# B&R Automation Studio project 8238 (part 24)

#### vc.ab
```automation-basic
;----------------------------------------------------
;Sequence 1 - SVC1 Vertical conveyor 1 D[900 + mySeq]
;----------------------------------------------------

PROGRAM _INIT
myHttp = 6
END_PROGRAM

PROGRAM _CYCLIC

;Inputs
myVC					    = 1 	;Vertical conveyor number
mySeq					    = 31		;Sequence number
myBag						= 319
myBufferBag					= 360
myIO						= 31
myZone						= 1
myFullLine					= 48
myFullBuffBag				= Line[myFullLine].FirstBag
myFullRelLine				= 0
myFullRelBag				= 0//Line[myFullRelLine].LastBag
myEmptyRelLine				= 0
myEmptyRelBag				= 0
myWeighBag					= 482

//Calculate weight
raw = DINT(AI1223[1])
raw = (raw * 2000)
Bag[myWeighBag].Cat = 1
IF (raw > 0) THEN
	Bag[myWeighBag].Wgt = UINT(raw/32767)
ELSE
	Bag[myWeighBag].Wgt = 0
ENDIF

IF (Bag[myWeighBag].Bid = 0) AND (BidStn > 0) THEN
	Bag[myWeighBag].Bid =  BidStn
	BidStn = 0
ENDIF

RB_PosnName[myVC].Name[1]	= posnNameHighLevelBagOut
RB_PosnName[myVC].Extra[1]	= posnExtraNone
RB_PosnName[myVC].Name[2]	= posnNameHighLevelBagIn
RB_PosnName[myVC].Extra[2]	= posnExtraNone
RB_PosnName[myVC].Name[3]	= posnNameLowLevelBagOut
RB_PosnName[myVC].Extra[3]	= posnExtraNone
RB_PosnName[myVC].Name[4]	= posnNameLowLevelBagIn
RB_PosnName[myVC].Extra[4]	= posnExtraNone

stopZone 		= Std.HaltSysZone[myZone] ;OR ;ZoneControl[myZone].requestAccess
;;ZoneControl[myZone].sequenceRunning[mySeq] = FALSE

I_BagAtOutbuffer			= FALSE
I_OutbufferOpen				= FALSE

;Set rail alignment direction
RailAlignPosn[1] 			= AlignRelease 	;Empty In
RailAlignPosn[2] 			= AlignReceive 	;Full Out
RailAlignPosn[3] 			= AlignRelease 	;Empty Out
RailAlignPosn[4] 			= AlignReceive 	;Full In
RailAlignPosn[5] 			= AlignNone
RailAlignPosn[6] 			= AlignNone

;Sequence Inputs
I_BagOnCarr					= X[myIO].X05
I_BagArriveCarr				= X[myIO].X04
I_PowerSave					= FALSE
I_BagAtFullBuffer			= Line[myFullLine].BufferProximity
I_BagReleased				= X[myIO + 1].X02// Released at high level
;BulkMode = NOT I_AutoMode

O_OpenBuffer					= FALSE
O_OpenCarrStop					= FALSE
O_Lamp                      	= FALSE
O_OpenFullBagBuffer				= FALSE

Request.VC[myVC]				= FALSE
Request.VC_HighLevel[myVC]  	= FALSE
Request.VC_LowLevel[myVC]	    = FALSE
RequestRel.VC_HighLevel[myVC]	= FALSE
RequestRel.VC_LowLevel[myVC]	= FALSE

EnableRel.PN[31]				= FALSE

;Lifting
strcpy(ADR(LiftIn.sDevice),ADR("SS1.IF1"))
strcpy(ADR(LiftIn.sParTblName),ADR("Param_1_5k"))
LiftIn.Node					= (10 + myVC)

LiftIn.DisableDrive			= FALSE
LiftIn.DoRef 				= FALSE
LiftIn.JogForwards 			= FALSE
LiftIn.JogReverse 			= FALSE
LiftIn.EStop				= Std.HaltSysZone[myZone]
LiftIn.PosnReq				= 0
LiftIn.MaxSpeed				= RB_Posn[myVC].Lift.MaxSpeed
LiftIn.PowerSave 			= FALSE
LiftIn.I_ForwardLimitOk		= X[myIO + 1].X01 	;Top limit   	- Do NOT Change to N.O.
LiftIn.I_ReverseLimitOk		= X[myIO + 1].X03	;Bottom limit	- Do NOT Change to N.O.
LiftIn.I_RefPosn			= X[myIO + 1].X04
LiftIn.I_RailOkRelease		= X[myIO].X07
LiftIn.I_RailOkReceive		= X[myIO].X06

LiftOut						= RB[myVC].Lift.SeqOut ;Copy drive outputs to local

;Shared Lift & Rotate
DisableDrive				= FALSE
RunMotor 					= FALSE
RunPosition					= 0

;Clear Interlock Signals
LOOP Posn = 1 TO 5 DO
	VCiLock[myVC].Posn[Posn].EnabSend 	= FALSE
ENDLOOP

Alarm[mySeq].Name 			= 0
Alarm[mySeq].Bag			= myBag
Alarm[mySeq].Beacon			= TRUE
Alarm[mySeq].Extra			= 0
Alarm[mySeq].Time			= 6000

;Setup Sequence
STEP = D[900 + mySeq]
;Setup Pulse contact
PLS = (STEP <> LASTSTEP)
LASTSTEP = STEP

;Sequence
IF (STEP = 0) THEN
	;Disabled
	DisableDrive 	= TRUE
ENDIF

;Combine Lift and Rotate into a single variable
DrivesReady		= LiftOut.RefComplete
DriveDisabled 	= (NOT PLS AND LiftOut.DriveDisabled) OR DebugMode
PosnOk	 		= (NOT PLS AND LiftOut.PosnOk)
RailOkReceive	= LiftIn.I_RailOkReceive
RailOkRelease	= LiftIn.I_RailOkRelease

;Power Save mode
IF I_PowerSave THEN
	LiftIn.PowerSave 	= TRUE
	LiftIn.MaxSpeed		= 300
ENDIF

;Carriage Empty Decide what to do next.
IF (STEP = 1) THEN
	;Cycle Count
    ;ZoneControl[myZone].sequenceRunning[mySeq] = TRUE
	IF PLS THEN
		CycleCount 						= CycleCount + 1
		RB_Perm[myVC].Lift.CycleCount 	= RB_Perm[myVC].Lift.CycleCount + 1
	ENDIF
	IF NOT Std.HaltSysZone[myZone]  THEN
		IF (CycleCount >= 500) THEN
			;If Referencing required then set 'Do Reference'
			;Put the sequence to a position step to enable the carriage
			;to retuen to the correct place after referencing
			LiftIn.DoRef 	= TRUE
			CycleCount 		= 0
		ELSE
			INC Count[mySeq]
			D[900 + mySeq] = 2
		ENDIF
	ENDIF
ENDIF

;Step 2. Move to empty bag in high level.....
IF (STEP = 2) THEN
	RunPosition	= POS_EMPTY_BAG_IN
	;ZoneControl[myZone].sequenceRunning[mySeq] = TRUE
	RunMotor	= (NOT Std.HaltSysZone[myZone] AND DrivesReady)
	IF PosnOk THEN
		D[900 + mySeq] = 3
	ENDIF
	IF (NOT Std.HaltSysZone[myZone] AND DrivesReady) THEN
		Alarm[mySeq].Name = almCarriageMoveFault
	ENDIF
ENDIF

GetFullBag	 = (Bag[myFullBuffBag].Cat > 0)
GetEmpty	 = RequestRel.PN[31] //And check lower loop space.

;Decide what to do
TON_10ms((NOT I_BagArriveCarr AND NOT I_BagOnCarr),300,CarriageClear,CarriageClearET)
IF (STEP = 3) THEN
	DisableDrive = TRUE
	IF CarriageClear AND (Bag[myBag].Cat = 0) AND NOT stopZone  THEN
	 	Request.VC[myVC] = TRUE // Tell CP31 that vc is in position..
		IF GetEmpty THEN
			D[900 + mySeq] = 4
		ELSE IF GetFullBag THEN
			D[900 + mySeq] = 9
		ENDIF
	ENDIF
  IF NOT CarriageClear THEN
		Alarm[mySeq].Name = almSwitchFault
	ELSE IF (Bag[myBag].Cat > 0) THEN
		Alarm[mySeq].Name = almBagDataError
	ENDIF
ENDIF

;Enable CP31 to release a bag
IF (STEP = 4) THEN
	DisableDrive = TRUE
    ;ZoneControl[myZone].sequenceRunning[mySeq] = TRUE
	EnableRel.PN[31] = (Bag[myBag].Cat = 0)
	IF (I_BagOnCarr OR I_BagArriveCarr) THEN
		D[900 + mySeq] = 5
	ENDIF
	IF NOT RailOkReceive THEN
		Alarm[mySeq].Name = almRailNotAligned
		Alarm[mySeq].Time = 100
	ENDIF
ENDIF

;Bag settles on carriage
TON_10ms(I_BagOnCarr,300,SettledCarriage,SettledCarriageET)
IF (STEP = 5) THEN
	DisableDrive = TRUE
	IF SettledCarriage AND (Bag[myBag].Cat > 0) AND NOT stopZone AND NOT EnableRel.VC_LowLevel[myVC] THEN
		D[900 + mySeq] = 6
	ELSE IF NOT SettledCarriage	THEN
		Alarm[mySeq].Name = almBagNotSettled
		Alarm[mySeq].Time = 9000
	ELSE IF (Bag[myBag].Cat = 0) THEN
		Alarm[mySeq].Name = ALM_BAG_DATA_ERROR
		Alarm[mySeq].Time = 0
	ENDIF
ENDIF

;Move carriage to empty bag out.
IF (STEP = 6) THEN
	RunPosition	= POS_EMPTY_BAG_OUT
    ;ZoneControl[myZone].sequenceRunning[mySeq] = TRUE
	RunMotor	= (NOT Std.HaltSysZone[myZone] AND DrivesReady)
	IF PosnOk THEN
		D[900 + mySeq] = 7
	ENDIF
	IF (NOT Std.HaltSysZone[myZone] AND DrivesReady) THEN
		Alarm[mySeq].Name = almCarriageMoveFault
	ENDIF
ENDIF

;Request Release
releaseValid = (Bag[myBag].Cat > 0)AND RailOkRelease
IF (STEP = 7) THEN
	DisableDrive = TRUE
	RequestRel.VC_LowLevel[myVC] = releaseValid
	IF EnableRel.VC_LowLevel[myVC] AND releaseValid THEN
		D[900 + mySeq] = 8
	ELSE IF NOT RailOkRelease THEN
		Alarm[mySeq].Name = almRailNotAligned
		Alarm[mySeq].Time = 100
	ELSE IF (Bag[myBag].Cat = 0) THEN
		Alarm[mySeq].Name = ALM_BAG_DATA_ERROR
		Alarm[mySeq].Time = 0
	ENDIF
ENDIF

;STEP 8 release empty bag
IF (STEP = 8) THEN
	DisableDrive = TRUE
	O_OpenCarrStop = releaseValid
	IF (Bag[myBag].Cat = 0) AND NOT EnableRel.VC_LowLevel[myVC] THEN
		IF GetFullBag OR (D[901] > 6) THEN//CHeck if there is a full bag, or the loading unit is releasing before moving back to the top,,
			D[900 + mySeq] = 9
		ELSE
			D[900 + mySeq] = 1
		ENDIF
	ELSE IF releaseValid THEN
		Alarm[mySeq].Name = ALM_BAG_NOT_RELEASED
	ELSE IF NOT RailOkRelease THEN
		Alarm[mySeq].Name = almRailNotAligned
		Alarm[mySeq].Time = 100
	ELSE IF (Bag[myBag].Cat = 0) THEN
		Alarm[mySeq].Name = ALM_BAG_DATA_ERROR
		Alarm[mySeq].Time = 0
	ENDIF
ENDIF

;Step 9. Move to full bag in.....
IF (STEP = 9) THEN
	RunPosition	= POS_FULL_BAG_IN
    ;ZoneControl[myZone].sequenceRunning[mySeq] = TRUE
	RunMotor	= (NOT Std.HaltSysZone[myZone] AND DrivesReady)
	IF PosnOk THEN
		D[900 + mySeq] = 10
	ENDIF
	IF (NOT Std.HaltSysZone[myZone] AND DrivesReady) THEN
		Alarm[mySeq].Name = almCarriageMoveFault
	ENDIF
ENDIF

//Wait for bag at full buffer
TON_10ms(I_BagAtFullBuffer,300,SettledFullBuffer,SettledFullBufferET)
IF (STEP = 10) THEN
	IF SettledFullBuffer AND (Bag[myBag].Cat = 0) AND (Bag[myFullBuffBag].Cat > 0) AND RailOkReceive THEN
		D[900 + mySeq] = 11
	ELSE IF NOT RailOkReceive THEN
		Alarm[mySeq].Name = ALM_RAIL_NOT_ALIGNED
		Alarm[mySeq].Time = 0
	ELSE IF (Bag[myBag].Cat > 0) THEN
		Alarm[mySeq].Name = ALM_BAG_DATA_ERROR
		Alarm[mySeq].Time = 0
	ELSE IF SettledFullBuffer AND (Bag[myFullBuffBag].Cat = 0) THEN
		Alarm[mySeq].Name = ALM_BAG_DATA_ERROR
		Alarm[mySeq].Bag = myFullBuffBag
	ELSE IF NOT SettledFullBuffer AND (Bag[myFullBuffBag].Cat > 0)THEN
		Alarm[mySeq].Name = ALM_BAG_NOT_SETTLED
		Alarm[mySeq].Time = 500
	ENDIF
ENDIF

;Open Full buffer stop
IF (STEP = 11) THEN
	DisableDrive = TRUE
    O_OpenFullBagBuffer = (Bag[myBag].Cat = 0) AND (Bag[myFullBuffBag].Cat > 0);
	IF I_BagOnCarr OR I_BagArriveCarr THEN
		Bag[myBag] = Bag[myFullBuffBag]
		Bag[myFullBuffBag] = Bag[0]
		D[900 + mySeq] = 12
	ENDIF
	IF (Bag[myBag].Cat > 0) THEN
		Alarm[mySeq].Name = ALM_BAG_DATA_ERROR
		Alarm[mySeq].Time = 0
	ELSE IF NOT RailOkReceive THEN
		Alarm[mySeq].Name = almRailNotAligned
		Alarm[mySeq].Time = 100
	ENDIF
ENDIF

;Bag settles on carriage
TON_10ms((STEP = 12) AND I_BagOnCarr AND NOT I_BagArriveCarr,300,SettledCarriage12,SettledCarriage12ET)
TON_10ms(((STEP = 12) AND (Bag[myWeighBag].Wgt < 1250)),600,weightOk,weightOkET)
IF (STEP = 12) THEN
	DisableDrive = TRUE
	IF SettledCarriage12 AND weightOk AND (Bag[myBag].Cat > 0) AND NOT stopZone  THEN
		Bag[myBag].Wgt := Bag[myWeighBag].Wgt;
		D[900 + mySeq] = 13
	ELSE IF NOT weightOk THEN
		Alarm[mySeq].Name = almBagOverWeight
	ELSE IF (Bag[myBag].Cat = 0) THEN
	//	Alarm[mySeq].Name = almBagDataError
	ELSE IF NOT stopZone THEN
		Alarm[mySeq].Name = almBagNotSettled
		Alarm[mySeq].Time = 9000
	ENDIF
ENDIF

;Move carriage to full bag out.
IF (STEP = 13) THEN
	RunPosition	= POS_FULL_BAG_OUT
    ;ZoneControl[myZone].sequenceRunning[mySeq] = TRUE
	RunMotor	= (NOT Std.HaltSysZone[myZone] AND DrivesReady)
	IF PosnOk THEN
		D[900 + mySeq] = 14
	ENDIF
	IF (NOT Std.HaltSysZone[myZone] AND DrivesReady) THEN
		Alarm[mySeq].Name = almCarriageMoveFault
	ENDIF
ENDIF

//Weighing step  Send to Data base. Add to batch...
IF (STEP = 14) THEN
	IF (Bag[myBag].Mis > 0) THEN
		_httpRequest
		IF httpComplete AND NOT EnableRel.VC_HighLevel[myVC] THEN
			myReportStn = 1
			IF (ReportLoading[myReportStn].Cat = 0) THEN
				ReportLoading[myReportStn].Prg := Bag[myBag].Prg;
				ReportLoading[myReportStn].Cat := Bag[myBag].Cat;
				ReportLoading[myReportStn].Cus := Bag[myBag].Cus;
				ReportLoading[myReportStn].Wgt := Bag[myBag].Wgt;
				ReportLoading[myReportStn].Cnt := 0;
				ReportLoading[myReportStn].Stn := myReportStn;
				ReportLoading[myReportStn].Mcn := 0;
				ReportLoading[myReportStn].Bid := Bag[myBag].Bid;
				ReportLoading[myReportStn].Mis := Bag[myBag].Mis;
				ReportLoading[myReportStn].TimeStamp := Bag[myBag].Timestamp;
				D[900 + mySeq] = 15
			ENDIF;
		ELSE
			Alarm[mySeq].Name = ALM_GENERAL_SEQUENCE
		ENDIF
	ELSE
		Alarm[mySeq].Name = ALM_BAG_DATA_ERROR
	ENDIF
ELSE
	httpComplete = 0
	HTTP_Comm[myHttp].Status = HTTP_COMM_STATUS_DISABLED
ENDIF;

DataValid = (Bag[myBag].Cat > 0)// AND (Bag[myFullRelBag].Cat = 0))
;check data valid
IF (STEP = 15) THEN
	DisableDrive = TRUE
	RequestRel.VC_HighLevel[myVC] = DataValid AND RailOkRelease AND NOT stopZone
	IF  EnableRel.VC_HighLevel[myVC] THEN
		D[900 + mySeq] = 16
	ELSE IF (Bag[myBag].Cat = 0) THEN
	//	Alarm[mySeq].Name = almBagDataError
	ELSE IF NOT RailOkRelease THEN
		Alarm[mySeq].Name = almRailNotAligned
		Alarm[mySeq].Time = 100
	ENDIF
ENDIF

;STEP 15 Open Stops release full bag
IF (STEP = 16) THEN
	DisableDrive = TRUE
    ;ZoneControl[myZone].sequenceRunning[mySeq] = TRUE
	O_OpenCarrStop = EnableRel.VC_HighLevel[myVC] AND RailOkRelease
	IF (NOT EnableRel.VC_HighLevel[myVC] OR I_BagReleased) AND (Bag[myBag].Cat = 0) THEN
		D[900 + mySeq] = 1
	ENDIF
	IF NOT stopZone THEN
		IF NOT EnableRel.VC_HighLevel[myVC]  AND (Bag[myBag].Cat > 0) THEN
			Alarm[mySeq].Name = ALM_BAG_DATA_ERROR
		ELSE IF NOT RailOkRelease THEN
			Alarm[mySeq].Name = almRailNotAligned
			Alarm[mySeq].Time = 100
		ENDIF
	ENDIF
ENDIF

;-----------------------------------------------------------
;No Changes required below here except PLC outputs at bottom
;-----------------------------------------------------------

;Positions Required
IF (RunPosition > 0) THEN
	LiftIn.PosnReq		= RB_Posn[myVC].Lift.Posn[RunPosition]
	LiftIn.RailAlign 	= RailAlignPosn[RunPosition]

	RotateIn.PosnReq	= RB_Posn[myVC].Rotate.Posn[RunPosition]
	RotateIn.RailAlign 	= RailAlignPosn[RunPosition]
ELSE
	LiftIn.PosnReq		= 0
	LiftIn.RailAlign	= 0

	RotateIn.PosnReq	= 0
	RotateIn.RailAlign 	= 0
ENDIF

;Bag detected on carriage at wrong time during operation
IF ((RunPosition > 0) AND RunMotor) THEN
	IF I_BagArriveCarr THEN
		LiftIn.EStop	= TRUE ;Force Quickstop
		RunPosition		= 0
		RunMotor		= FALSE
		D[900 + mySeq] 	= 97
	ELSE IF (I_BagOnCarr AND (RailAlignPosn[RunPosition] = AlignReceive)) THEN
		LiftIn.EStop	= TRUE ;Force Quickstop
		RunPosition		= 0
		RunMotor		= FALSE
		D[900 + mySeq] 	= 98
	ENDIF
ENDIF
IF (STEP = 97) THEN
	DisableDrive = TRUE
	Alarm[mySeq].Name 	= almDisableSequence
	Alarm[mySeq].Time			= 100
ENDIF
IF (STEP = 98) THEN
	DisableDrive = TRUE
	Alarm[mySeq].Name 	= almDisableSequence
	Alarm[mySeq].Time			= 100
ENDIF

;Position Setup
TON_10ms(VCHeartBeat = D[84],100,VCActionDisabled,VCActionDisabledET)
IF (STEP = 99) THEN

	RB_Posn[myVC].Lift.OperationMode 	= 1 ;Manual Position Setup
	RB_Posn[myVC].Rotate.OperationMode 	= 1 ;Manual Position Setup

	;Read values sent from TrackView
	VCIndex 	= D[81]
	VCMode 		= D[82]
	VCAction 	= D[83]
	VCHeartBeat = D[84]

	IF ((VCIndex = myVC) AND NOT VCActionDisabled) THEN

		IF (VCMode = ModeReference) THEN
			LiftIn.DoRef 			= TRUE
			RotateIn.DoRef 			= TRUE
		ELSE IF (VCMode = ModeManualMove) THEN
			LiftIn.JogForwards 		= (VCAction = ActionMoveUp)
			LiftIn.JogReverse 		= (VCAction = ActionMoveDown)
			RotateIn.JogReverse		= (VCAction = ActionMoveLeft)
			RotateIn.JogForwards	= (VCAction = ActionMoveRight)
		ELSE IF (VCMode = ModePosnTune) THEN
			AutoTuneSequence		= 1
			AutoTunePosition		= VCAction
		ELSE IF (VCMode = ModeMovePosn) THEN
			RunMotor				= (NOT Std.HaltSysZone[myZone] AND DrivesReady); AND ;PositionSetup)
			LiftIn.MaxSpeed 		= 200
			RotateIn.MaxSpeed 		= 200
			IF (VCAction = 100) THEN
				LiftIn.PosnReq 		= RB_Posn[myVC].Lift.RefOffset
				RotateIn.PosnReq 	= RB_Posn[myVC].Rotate.RefOffset
			ELSE
				LiftIn.PosnReq		= RB_Posn[myVC].Lift.Posn[VCAction]
				RotateIn.PosnReq	= RB_Posn[myVC].Rotate.Posn[VCAction]
			ENDIF
		ENDIF

	ENDIF

	;Auto Position Tune Sequnece
	;---------------------------
	IF (AutoTuneSequence = 1) THEN
		;Wait for release of Autotune Button / Command
		IF (VCMode <> ModePosnTune) THEN
			AutoTuneSequence = 2
		ENDIF
	ELSE IF (AutoTuneSequence = 2) THEN
		;Check if rail Aligned
		Aligned = (((RailAlignPosn[AutoTunePosition] = AlignReceive) AND LiftIn.I_RailOkReceive) OR ((RailAlignPosn[AutoTunePosition] = AlignRelease) AND LiftIn.I_RailOkRelease))
		;Begin Lift Tune
		IF Aligned THEN
			LiftIn.AutoTunePosn		= AutoTunePosition
			LiftIn.AutoTuneReceive 	= (RailAlignPosn[AutoTunePosition] = AlignReceive)
			IF (LiftOut.AutoTunePosn = AutoTunePosition) THEN
				AutoTuneSequence = 3
			ENDIF
		ELSE
			AutoTuneSequence = 0 ;Cancel Auto Tune
		ENDIF
	ELSE IF (AutoTuneSequence = 3) THEN
		;Wait for Lift to complete Tune
		IF (LiftOut.AutoTunePosn = 0) THEN
			AutoTuneSequence = 4
		ENDIF
	ELSE IF (AutoTuneSequence = 4) THEN
		;Move to new position
		LiftIn.AutoTunePosn		= 0 ;Cancel Tune
		RunMotor				= (NOT Std.HaltSysZone[myZone] AND DrivesReady); AND ;PositionSetup)
		LiftIn.MaxSpeed 		= 200
		RotateIn.MaxSpeed		= 0  ;Don't allow rotate to move
		LiftIn.PosnReq			= RB_Posn[myVC].Lift.Posn[AutoTunePosition]
		RotateIn.PosnReq		= 0
		IF LiftOut.PosnOk THEN
			AutoTuneSequence = 5
		ENDIF
	ELSE IF (AutoTuneSequence = 5) THEN
		;Begin Rotate Tune
		RotateIn.AutoTunePosn 		= AutoTunePosition
		RotateIn.AutoTuneReceive 	= (RailAlignPosn[AutoTunePosition] = AlignReceive)
		IF (RotateOut.AutoTunePosn = AutoTunePosition) THEN
			AutoTuneSequence = 6
		ENDIF
	ELSE IF (AutoTuneSequence = 6) THEN
		;Wait for Rotate to complete Tune
		IF (RotateOut.AutoTunePosn = 0) THEN
			AutoTuneSequence = 7
		ENDIF
	ELSE IF (AutoTuneSequence = 7) THEN
		;Move to new position
		RotateIn.AutoTunePosn	= 0 ;Cancel Tune
		RunMotor				= (NOT Std.HaltSysZone[myZone] AND DrivesReady); AND ;PositionSetup)
		LiftIn.MaxSpeed 		= 0
		RotateIn.MaxSpeed		= 200
		LiftIn.PosnReq			= 0
		RotateIn.PosnReq		= RB_Posn[myVC].Rotate.Posn[AutoTunePosition]
		IF RotateOut.PosnOk THEN
			AutoTuneSequence = 0
		ENDIF
	ENDIF

ELSE
	;Set Operation mode to Normal
	RB_Posn[myVC].Lift.OperationMode 	= 0
	RB_Posn[myVC].Rotate.OperationMode 	= 0
	;Cancel Auto Tune
	AutoTuneSequence 					= 0
	LiftIn.AutoTunePosn 				= 0
	RotateIn.AutoTunePosn 				= 0
ENDIF

;Lift Drive Alarms
IF (LiftOut.Status = FC302_SEQ_RefNotFound) THEN
	Alarm[mySeq].Name = almLiftRefNotFound
	Alarm[mySeq].Time = 10
ELSE IF (LiftOut.Status = FC302_SEQ_ParameterError) THEN
	Alarm[mySeq].Name = almLiftParameterError
	Alarm[mySeq].Time = 10
ELSE IF (LiftOut.Status = FC302_SEQ_RefSwitchFault) THEN
	Alarm[mySeq].Name = almLiftRefSwitchFault
	Alarm[mySeq].Time = 10
ELSE IF (LiftOut.Status = FC302_SEQ_ReleaseSwitchFault) THEN
	Alarm[mySeq].Name = almReleaseSwitchFault
	Alarm[mySeq].Time = 10
ELSE IF (LiftOut.Status = FC302_SEQ_ReceiveSwitchFault) THEN
	Alarm[mySeq].Name = almReceiveSwitchFault
	Alarm[mySeq].Time = 10
ELSE IF (LiftOut.Status = FC302_SEQ_RailNotAligned) THEN
	Alarm[mySeq].Name = almReleaseSwitchFault
	Alarm[mySeq].Time = 10
ENDIF

;Inputs to drive control sequence
LiftIn.Run			     	= RunMotor
LiftIn.DisableDrive 	= DisableDrive
RB[myVC].Lift.SeqIn 	= LiftIn 	;Copy local to drive inputs

TON_10ms(NOT Std.HaltSysZone[myZone],100,HaltSysZoneClear,HaltSysZoneClearET)	; Safe zone
OpenStopEnabled = (HaltSysZoneClear AND LiftOut.DriveDisabled)

;-----------------------------------
;PLC Outputs - adjust to suit system
;-----------------------------------
Y[22].Y05 = (RailOkReceive AND ((STEP = 11) OR (STEP = 12)) AND DriveDisabled)  ; Safety Stop Low level
Y[myIO + 1].Y05 = (RailOkReceive AND ((STEP = 3) OR (STEP = 4) OR (STEP = 5)) AND DriveDisabled) ; Safety Stop High level
Y[4].Y06 		= (O_OpenCarrStop AND RailOkRelease AND OpenStopEnabled AND DriveDisabled)

Line[myFullLine].BufferStop := O_OpenFullBagBuffer

;Don't allow forcing of carriage movement and carriage stop
YForceDisable[myIO].Y07 	= TRUE
YForceDisable[myIO].Y08 	= TRUE
;YForceDisable[6].Y04 	= TRUE

;Alarms
TimerAlarm.IN 		= NOT PLS AND (Alarm[mySeq].Name > 0)
TimerAlarm.PT 		= Alarm[mySeq].Time
TimerAlarm FUB TON_10ms()
Alarm[mySeq].On 	= TimerAlarm.Q
Alarm[mySeq].ET 	= TimerAlarm.ET

END_PROGRAM
```

#### _httpRequest.st
```iecst
ACTION _httpRequest:

	CASE HTTP_Comm[myHttp].Status OF

		HTTP_COMM_STATUS_DISABLED:

			//Build Request String..
			requestURL := HTTP_IF_CALL_USP_NOREPLY_URL;
			itoa(Bag[myBag].Mis,ADR(batchString));
			itoa(Bag[myWeighBag].Wgt,ADR(weightString));
			//Bag[myBag].Wgt := Bag[myWeighBag].Wgt;

			requestData := CONCAT(HTTP_POST_BATCH_UPDATE_DRY_WGT,'@BatchID_Int=');
			requestData := CONCAT(requestData,batchString);
			requestData := CONCAT(requestData,',@DryWeight=');
			requestData := CONCAT(requestData,weightString);

			HTTP_Comm[myHttp].Command.Method := httpMETHOD_POST;
			HTTP_Comm[myHttp].Command.Cmd_URL.Adr := ADR(requestURL);
			HTTP_Comm[myHttp].Command.Cmd_URL.Size := LEN(requestURL);
			HTTP_Comm[myHttp].Command.Body_Data.Adr := ADR(requestData);
			HTTP_Comm[myHttp].Command.Body_Data.Size := strlen(ADR(requestData));
			HTTP_Comm[myHttp].Command.ResponseData.Adr := 0;
			HTTP_Comm[myHttp].Command.ResponseData.Size := 0;
			HTTP_Comm[myHttp].Status := HTTP_COMM_STATUS_ACTIVE_WAIT_BUF;

		HTTP_COMM_STATUS_ACTIVE_WAIT_BUF:
		//Command is sent to ring buffer.
		HTTP_COMM_STATUS_IN_BUFFER:
		//Command recieved and in ring buffer
		HTTP_COMM_STATUS_IN_PROCESS:
		//Command being processed by httpClient.
		HTTP_COMM_STATUS_COMPLETE:
			httpComplete := 1;
			//HTTP_Comm[myHttp].Status := HTTP_COMM_STATUS_DISABLED;
		HTTP_COMM_STATUS_ERROR: // Go to next index
			HTTP_Comm[myHttp].Status := HTTP_COMM_STATUS_DISABLED;

	END_CASE;

END_ACTION
```

### Program Logical/Robo_Drive_Control/Lift_v8_1 (IEC, version 8.00.2)

#### Lift.var - Local variables
```iecst
(********************************************************************
 * COPYRIGHT --
 ********************************************************************
 * Program: PosnVC
 * File: PosnVC.var
 * Author: D.Jefferys
 * Created: February 12, 2009
 ********************************************************************
 * Local variables of program PosnVC
 ********************************************************************)
VAR
	AutoNewPosn : DINT;
	AutoPosnDiff : DINT;
	AutoSavedBottom : DINT;
	AutoSavedTop : DINT;
	CANopenNMT_0 : CANopenNMT;
	DisableDrive : BOOL;
	DistRemain : DINT;
	EnableDrive : BOOL;
	EnableForwards : BOOL;
	EnableReference : BOOL;
	EnableReverse : BOOL;
	EnableTune : BOOL;
	FC302_ReadParam_0 : FC302_ReadParam;
	FC302_ReadParamTbl_0 : FC302_ReadParamTbl;
	FC302_ReadSTW_0 : FC302_ReadSTW;
	FC302_WriteCTW_0 : FC302_WriteCTW;
	FC302_WriteParam_0 : FC302_WriteParam;
	I_InPosition : BOOL;
END_VAR
VAR RETAIN
	idx : UINT;
END_VAR
VAR
	LimitsOk : BOOL;
	ManualControl : BOOL;
	MaxHz : UINT;
	MonitorIndex : UINT := 0;
	MonitorSubIndex : USINT;
	MotorNomHz : UINT;
	myRead : UDINT;
	myStatus : UINT;
	node : USINT;
	ParameterEnable : BOOL;
	PosnDiff : DINT;
	PosnValid : BOOL;
	PowerSave : BOOL;
	QuickStop : BOOL;
	RailAligned : BOOL;
	RampDist : REAL;
	RampFactor : REAL;
	RampTime : UINT;
	Referencing : BOOL;
	ReleaseSwitchOk : BOOL := FALSE;
	ReceiveSwitchOk : BOOL := FALSE;
	RequiredHz : UINT;
	ResetTrip : BOOL;
	RunSpeed : REAL;
	RunTask : BOOL;
	SavedBottom : DINT;
	SavedPosition : DINT;
	SavedTop : DINT;
	ScanClock : TIME;
	ScanCount : UINT;
	ScanLastClock : TIME;
	ScanNow : TIME := T#0ms;
	sDevice : STRING[12];
	SlowWindow : DINT;
	sTableName : STRING[10];
	STEP : UINT;
	StopDist : DINT;
	StopFactor : REAL;
	TableTooLarge : BOOL;
	TaskName : STRING[11];
	TaskNameID : UINT;
	TaskNameLen : UINT;
	TON_10ms_PastRef : TON_10ms;
	TON_10ms_Restart : TON_10ms;
	TON_10ms_Retry : TON_10ms;
	WriteIndex : UINT;
	WriteListLength : UINT;
	JogHz : UINT;
	TmrJog : TON_10ms;
	AlignSwitchCheck : BOOL;
	AlignSwitchesOk : BOOL;
	mySlowWindow : DINT;
	myDist : DINT;
	RefSpeed : UINT;
	CountCardFailedPLS : BOOL;
	RetryCount : UINT;
	I_RefPosnPLS : BOOL;
	AutoRefTolerance : DINT;
	Debug_PositionErrorCount : UDINT;
	PositionErrorLastValue : ARRAY[0..100] OF DINT;
	IndexPostion : UINT;
	Debug_CycleCount : UDINT;
	DebugLastActual : DINT;
	DebugRef : DINT;
	PositionError : DINT;
	TestValue : DINT;
	TestResult : DINT;
END_VAR
```

#### Lift.ab - Cyclic code
```automation-basic
;--------------------------------------
;Lift Drive Control - Original 2 Column
;--------------------------------------

;Version 1.00 23/02/2009 D.J. First Issue
;Version 2.00 03/11/2010 D.J. Changed RB to RB (Robo)
;Version 3.00 04/12/2010 D.J. New distance calculation by using encoder pulses for 1 meter
;Version 4.00 04/03/2011 D.J. Set RunHz to 0 when not on step 30
;Version 5.00 08/01/2013 T.R Add module OK to monitor Counter Card and force step 0 after error/powerup..Increased Param Count for Brake contact monitoring. Force init values when 0.
;Version 5.01 12/03/2013 T.R Change function of module OK monitoring to always restart seq after fail due to power cycles on remote panels.
;Version 6.01 			T.R Add Auto Reference function
;Version 6.02 27/11/2015 TR. Add Correct comments,
;Version V8 -- TR Send QS command when enable is off due to DANFOSS issues.

PROGRAM _INIT

 	;Set array index with each init call
	idx  = 0

	TaskNameID = ST_name(0,ADR(TaskName),0)

	IF (TaskNameID = 0) THEN
		TaskNameLen = strlen(ADR(TaskName))
		idx 		= UINT(atoi(ADR(TaskName) + (TaskNameLen - 1)))
	ENDIF

	RunTask = (idx > 0) and (idx <= (SIZEOF(RB)/SIZEOF(RB[0])))

	IF RunTask THEN

		;Calculate in future for different arrangements
		;----------------------------------------------

		;New calculation based on measuring the pulsed for 1000 mm of Travel
		;-------------------------------------------------------------------

		;Pulses per meter = 122864.6
		;My Ratio (Gearbox and Cog combined) = 4096 / 122.8646 = 33.3375
		;mm/minute 				= Motor Nominal Speed 1500 * My Ratio = 50006.25
		;mm/sec @ 50 Hz 		= 833.4375
		;mm/Hz 	833.4375 / 50 	= 16.6687

		RB[idx].Lift.PulsePer10th_mm = REAL(12.2865)
		RB[idx].Lift.mmPerHz = 16.6687
		;Force Init value if 0
		IF RB_Posn[idx].Lift.RefOffset = 0 THEN
			RB_Posn[idx].Lift.RefOffset = 20000 ; 2metres
		ENDIF
		IF RB_Posn[idx].Lift.MaxSpeed = 0 THEN
			RB_Posn[idx].Lift.MaxSpeed = 200
		ENDIF

		// Temp to force input parameters.

		strcpy(ADR(RB[idx].Lift.SeqIn.sDevice),ADR("SL1.IF3"))
		strcpy(ADR(RB[idx].Lift.SeqIn.sParTblName),ADR("Param_1_5k"))
		RB[idx].Lift.SeqIn.Node := 10 + USINT(idx);
		RB[idx].Lift.ModuleOK := TRUE
		// END

	ENDIF

	STEP 					= 0
	RB[idx].Lift.SeqStep	= 0
	RetryCount				= 0

END_PROGRAM
PROGRAM _CYCLIC

	;----
	;Lift
	;----

	myStatus = FC302_SEQ_OK

	;CAN node, Parameter Table Name and IF address
	node 	= RB[idx].Lift.SeqIn.Node
	strcpy(ADR(sTableName),ADR(RB[idx].Lift.SeqIn.sParTblName))
	strcpy(ADR(sDevice),ADR(RB[idx].Lift.SeqIn.sDevice))

	RB[idx].Lift.SeqIn.I_RefPosn  = X[30 + (idx * 2)].X04

	;Read drive status
	FC302_ReadSTW_0.StatusWord = RB[idx].Lift.CAN.StatusWord
	FC302_ReadSTW_0 FUB FC302_ReadSTW()
	RB[idx].Lift.STW = FC302_ReadSTW_0.STW

	;Clear control word - drive stopped
	RB[idx].Lift.CTW.ExtRefSelectionLSB 	= FALSE
	RB[idx].Lift.CTW.ExtRefSelectionMSB 	= FALSE
	RB[idx].Lift.CTW.DC_Brake				= FALSE
	RB[idx].Lift.CTW.Coasting				= FALSE
	RB[idx].Lift.CTW.QuickStop				= FALSE
	RB[idx].Lift.CTW.HoldOutputFreq			= FALSE
	RB[idx].Lift.CTW.RampStopStart			= FALSE
	RB[idx].Lift.CTW.ResetTrip				= ResetTrip
	RB[idx].Lift.CTW.Jog					= FALSE
	RB[idx].Lift.CTW.RampSelection			= FALSE
	RB[idx].Lift.CTW.DataValid				= TRUE
	RB[idx].Lift.CTW.Relay01Active			= FALSE
	RB[idx].Lift.CTW.Relay02Active			= FALSE
	RB[idx].Lift.CTW.ParaSetUpLSB			= FALSE
	RB[idx].Lift.CTW.ParaSetUpMSB			= FALSE
	RB[idx].Lift.CTW.Reverse				= FALSE

	RB[idx].Lift.RunForwards				= FALSE
	RB[idx].Lift.RunReverse					= FALSE
	RB[idx].Lift.CAN.TargetVelocity			= 0
	RB[idx].Lift.RunFreq 					= 0
	RB[idx].Lift.SeqOut.RefComplete 		= FALSE
	RB[idx].Lift.SeqOut.PosnOk				= FALSE
	RB[idx].Lift.SeqOut.DriveDisabled		= FALSE
	Referencing								= FALSE
	DisableDrive 							= (RB[idx].Lift.SeqIn.DisableDrive OR RB[idx].Lift.SeqIn.EStop OR NOT RB[idx].Lift.STW.DriveReady OR NOT RB[idx].Lift.ModuleOK)
	LimitsOk								= (RB[idx].Lift.SeqIn.I_ForwardLimitOk AND RB[idx].Lift.SeqIn.I_ReverseLimitOk)
	ManualControl							= (RB_Posn[idx].Lift.OperationMode = 1)

	;Init var ensure not lost if no Init
	RB[idx].Lift.PulsePer10th_mm 			= REAL(12.2865)
	RB[idx].Lift.mmPerHz 					= 16.6687

	;Current Position
	RB[idx].Lift.PosnActRaw = (RB[idx].Lift.Encoder + $7FFFFFFF)
	RB[idx].Lift.PosnAct	= DINT(RB[idx].Lift.PosnActRaw / RB[idx].Lift.PulsePer10th_mm)
	RB[idx].Lift.PosnNow	= ((RB_Retain[idx].Lift.PosnRef - RB[idx].Lift.PosnAct) + RB_Posn[idx].Lift.RefOffset)
	RB[idx].Lift.DistRemain = ABS(RB[idx].Lift.SeqIn.PosnReq - RB[idx].Lift.PosnNow)

	;TrackView Display
	RB_Posn[idx].Lift.PositionNow 	= RB[idx].Lift.PosnNow
	RB_Posn[idx].Lift.CycleCount 	= RB_Perm[idx].Lift.CycleCount

	;Step Shifting
	STEP = RB[idx].Lift.SeqStep
	RB_Posn[idx].Lift.SeqStep = DINT(STEP)

	;Enable Parameter writing slower speed - Every 60ms
	ScanClock 		= clock_ms()
	ScanNow 		= (ScanClock - ScanLastClock)
	ScanLastClock 	= ScanClock
	ScanCount 		= (ScanCount + UINT(ScanNow))
	IF (ScanCount >= 60) THEN
		ScanCount = 0
	ENDIF
	ParameterEnable = (ScanCount = 0)

	;If ModuleOK Fails force reference.// Change to restart to CAN Sequence to ensure full control and correct params
;	F_TRIG(RB[idx].Lift.ModuleOK,CountCardFailedPLS)
;	IF CountCardFailedPLS AND (RetryCount < 5) THEN
;		RetryCount = RetryCount + 1  ;If required limit number of retries on the reference TEST IF REQUIRED> HOW TO HANDLE ERROR??
;		RB[idx].Lift.SeqIn.DoRef = TRUE
;	ENDIF
	IF NOT RB[idx].Lift.ModuleOK THEN	; Code to disable drive if count card failed/poweroff.
		RB[idx].Lift.SeqStep = 0
	ENDIF

	;Step 0 ;Disabled
	IF (STEP = 0) THEN
		IF (RunTask AND RB[idx].Lift.ModuleOK) THEN
			RB[idx].Lift.SeqStep = 1
		ELSE
			;Do Nothing
		ENDIF
	ENDIF

	;Set CAN node to pre-operational
	TON_10ms_Restart.IN = (STEP = 1)
	TON_10ms_Restart.PT = 1000
	TON_10ms_Restart FUB TON_10ms()
	IF (STEP = 1) THEN

		IF (StartNode = node) THEN
			StartNode = 0
		ENDIF

		myStatus = FC302_SEQ_SetCANPreOperational

		IF (RB[idx].Lift.CAN.ModuleOk OR (RB[idx].Lift.CAN.NodeStatus = 3)) THEN

			CANopenNMT_0.enable 	= TRUE
			CANopenNMT_0.pDevice 	= ADR(sDevice)
			CANopenNMT_0.node 		= node
			CANopenNMT_0.state 		= coENTER_PRE_OPERATIONAL
			CANopenNMT_0 FUB CANopenNMT()

			IF (CANopenNMT_0.status = 0) OR (CANopenNMT_0.status < 65535) THEN
				RB[idx].Lift.SeqStep = 10
			ENDIF

		ELSE IF TON_10ms_Restart.Q THEN
			RB[idx].Lift.SeqStep = 2 ;Reset node here if not true
		ENDIF

	ENDIF

	;Restart node
	IF (STEP = 2) THEN

		myStatus = FC302_SEQ_RestartCANnode

		CANopenNMT_0.enable 	= TRUE
		CANopenNMT_0.pDevice 	= ADR(sDevice)
		CANopenNMT_0.node 		= node
		CANopenNMT_0.state 		= coRESET_NODE
		CANopenNMT_0 FUB CANopenNMT()

		IF (CANopenNMT_0.status = 0) OR (CANopenNMT_0.status < 65535) THEN
			RB[idx].Lift.SeqStep = 1
		ENDIF

	ENDIF

	;Read from parameter table
	IF (STEP = 10) THEN

		myStatus = FC302_SEQ_ReadParameterTable

		TableTooLarge = FALSE

		FC302_ReadParamTbl_0.Enable 		= TRUE
		FC302_ReadParamTbl_0.adrTableName 	= ADR(sTableName)
		FC302_ReadParamTbl_0.adrDestTable 	= ADR(RB[idx].Lift.ParaList)
		FC302_ReadParamTbl_0.ParamLimit 	= (SIZEOF(RB[idx].Lift.ParaList) / 8)
		FC302_ReadParamTbl_0 FUB FC302_ReadParamTbl()

		IF FC302_ReadParamTbl_0.Status = 0 THEN
			WriteListLength = FC302_ReadParamTbl_0.ParamCount	;Total parameters to write to the drive
			WriteIndex 		= 0 								;First index to write 0 not used
			RB[idx].Lift.SeqStep = 11
		ELSE IF FC302_ReadParamTbl_0.Status = 1 THEN
			TableTooLarge = TRUE
		ELSE
			;Error
		ENDIF

	ENDIF

	;Write parameter list to drive
	IF (STEP = 11) THEN

		myStatus = FC302_SEQ_WriteParameters

		IF ParameterEnable THEN

			FC302_WriteParam_0.enable 	= TRUE
			FC302_WriteParam_0.pDevice 	= ADR(sDevice)
			FC302_WriteParam_0.node 	= node
			FC302_WriteParam_0.index 	= RB[idx].Lift.ParaList[WriteIndex].index
			FC302_WriteParam_0.subindex = RB[idx].Lift.ParaList[WriteIndex].subindex
			FC302_WriteParam_0.data 	= RB[idx].Lift.ParaList[WriteIndex].data
			FC302_WriteParam_0.bytelen 	= RB[idx].Lift.ParaList[WriteIndex].datalen
			FC302_WriteParam_0 FUB FC302_WriteParam()

			IF (FC302_WriteParam_0.status = 0) THEN
				RB[idx].Lift.SeqStep = 12
			ENDIF

		ENDIF

	ENDIF

	;Read Parameter from drive
	IF (STEP = 12) THEN

		myStatus = FC302_SEQ_WriteParameters

		IF ParameterEnable THEN

			FC302_ReadParam_0.enable 	= TRUE
			FC302_ReadParam_0.pDevice 	= ADR(sDevice)
			FC302_ReadParam_0.node 		= node
			FC302_ReadParam_0.index 	= RB[idx].Lift.ParaList[WriteIndex].index
			FC302_ReadParam_0.subindex 	= RB[idx].Lift.ParaList[WriteIndex].subindex
			FC302_ReadParam_0 FUB FC302_ReadParam()

			IF (FC302_ReadParam_0.status = 0) THEN
				myRead 	= UDINT(FC302_ReadParam_0.data)
				IF RB[idx].Lift.ParaList[WriteIndex].data = myRead THEN
					WriteIndex = WriteIndex + 1
					;Once = all parameters have been completed as 60 = 0-59
					IF (WriteIndex = WriteListLength) THEN
						RB[idx].Lift.SeqStep = 13
					ELSE
						RB[idx].Lift.SeqStep = 11 ;Write Next Parameter
					ENDIF
				ELSE
					RB[idx].Lift.ParamWrite.ErrorCount 	= RB[idx].Lift.ParamWrite.ErrorCount + 1
					RB[idx].Lift.ParamWrite.Index 		= RB[idx].Lift.ParaList[WriteIndex].index
					RB[idx].Lift.ParamWrite.SubIndex 	= RB[idx].Lift.ParaList[WriteIndex].subindex
					RB[idx].Lift.SeqStep = 11 ;Try Write Again
				ENDIF
			ENDIF

		ENDIF

	ENDIF

	;Store Parameters
	IF (STEP = 13) THEN

		myStatus = FC302_SEQ_WriteParameters

		IF ParameterEnable THEN

			FC302_WriteParam_0.enable 	= TRUE
			FC302_WriteParam_0.pDevice 	= ADR(sDevice)
			FC302_WriteParam_0.node 	= node
			FC302_WriteParam_0.index 	= 1031
			FC302_WriteParam_0.subindex = 0
			FC302_WriteParam_0.data 	= 1
			FC302_WriteParam_0.bytelen 	= 1
			FC302_WriteParam_0 FUB FC302_WriteParam()

			IF (FC302_WriteParam_0.status = 0) THEN
				RB[idx].Lift.SeqStep = 14
			ENDIF

		ENDIF

	ENDIF

	;Check Parameters are stored
	IF (STEP = 14) THEN

		myStatus = FC302_SEQ_CheckParamStored

		IF ParameterEnable THEN

			FC302_ReadParam_0.enable 	= TRUE
			FC302_ReadParam_0.pDevice 	= ADR(sDevice)
			FC302_ReadParam_0.node 		= node
			FC302_ReadParam_0.index 	= 1031
			FC302_ReadParam_0.subindex 	= 0
			FC302_ReadParam_0 FUB FC302_ReadParam()

			IF (FC302_ReadParam_0.status = 0) THEN
				IF (FC302_ReadParam_0.data = 0) THEN
					RB[idx].Lift.SeqStep = 15
				ENDIF
			ENDIF

		ENDIF

	ENDIF

	;Start CAN node
	IF (STEP = 15) THEN

		IF (StartNode = 0) THEN
			StartNode = node
		ENDIF

		IF (ParameterEnable AND (StartNode = node)) THEN

			myStatus = FC302_SEQ_StartCANnode

			CANopenNMT_0.enable 	= TRUE
			CANopenNMT_0.pDevice 	= ADR(sDevice)
			CANopenNMT_0.node 		= node
			CANopenNMT_0.state 		= coSTART_REMOTE_NODE
			CANopenNMT_0 FUB CANopenNMT()

			IF (CANopenNMT_0.status = 0) THEN
				RB[idx].Lift.SeqStep = 20
			ENDIF
		ENDIF

	ENDIF

	;Wait for drive operational
	TON_10ms_Retry.IN = (STEP = 20)
	TON_10ms_Retry.PT = 100 ;2000
	TON_10ms_Retry FUB TON_10ms()
	IF (STEP = 20) THEN
		myStatus = FC302_SEQ_WaitDriveOperational
		IF RB[idx].Lift.CAN.ModuleOk THEN
			IF (StartNode = node) THEN
				StartNode = 0
			ENDIF
			RB[idx].Lift.SeqStep 	= 21
		ELSE IF TON_10ms_Retry.Q THEN
			IF (StartNode = node) THEN
				StartNode = 0
			ENDIF
			RB[idx].Lift.SeqStep 	= 15 ;0
		ENDIF
	ENDIF

	;-----------------
	;Find ref Position
	;-----------------

	EnableReference = NOT DisableDrive

	;Past Reference position timer
	TON_10ms_PastRef.IN = NOT RB[idx].Lift.SeqIn.I_RefPosn
	TON_10ms_PastRef.PT = 30
	TON_10ms_PastRef FUB TON_10ms()

	RefSpeed = 100 ;150 ;15Hz

	;Move carriage down until refence or bottom limit
	IF (STEP = 21) THEN
		myStatus = FC302_SEQ_Referencing
		Referencing					= TRUE
		RB[idx].Lift.RunForwards 	= FALSE
		RB[idx].Lift.RunReverse 	= EnableReference
		RB[idx].Lift.RunFreq		= RefSpeed
		IF RB[idx].Lift.SeqIn.I_RefPosn THEN
			RB[idx].Lift.SeqStep = 23
		ELSE IF NOT RB[idx].Lift.SeqIn.I_ReverseLimitOk THEN
			RB[idx].Lift.SeqStep = 22
		ELSE IF NOT RB[idx].Lift.SeqIn.I_ForwardLimitOk THEN
			myStatus = FC302_SEQ_MotorWiringFault
		ENDIF
	ENDIF

	;Bottom limit was found - try moving up
	IF (STEP = 22) THEN
		myStatus = FC302_SEQ_Referencing
		Referencing					= TRUE
		RB[idx].Lift.RunForwards 	= EnableReference
		RB[idx].Lift.RunReverse 	= FALSE
		RB[idx].Lift.RunFreq		= RefSpeed
		IF RB[idx].Lift.SeqIn.I_RefPosn THEN
			RB[idx].Lift.SeqStep = 23
		ELSE IF NOT RB[idx].Lift.SeqIn.I_ForwardLimitOk THEN
			myStatus = FC302_SEQ_RefNotFound
		ENDIF
	ENDIF

	;Move carriage down past reference
	IF (STEP = 23) THEN
		myStatus = FC302_SEQ_Referencing
		Referencing					= TRUE
		RB[idx].Lift.RunForwards 	= FALSE
		RB[idx].Lift.RunReverse 	= EnableReference
		RB[idx].Lift.RunFreq		= RefSpeed
		IF TON_10ms_PastRef.Q THEN
			RB[idx].Lift.SeqStep = 24
		ENDIF
	ENDIF

	;Move carriage back up to reference
	IF (STEP = 24) THEN
		myStatus = FC302_SEQ_Referencing
		Referencing					= TRUE
		RB[idx].Lift.RunForwards 	= EnableReference
		RB[idx].Lift.RunReverse 	= FALSE
		RB[idx].Lift.RunFreq		= RefSpeed
		IF RB[idx].Lift.SeqIn.I_RefPosn THEN
			RB[idx].Lift.SeqStep = 25
		ENDIF
	ENDIF

	;Move carriage up clear of reference
	IF (STEP = 25) THEN
		myStatus = FC302_SEQ_Referencing
		Referencing					= TRUE
		RB[idx].Lift.RunForwards 	= EnableReference
		RB[idx].Lift.RunReverse 	= FALSE
		RB[idx].Lift.RunFreq		= 100
		IF TON_10ms_PastRef.Q THEN
			RB[idx].Lift.SeqStep = 26
		ENDIF
	ENDIF

	;Move carriage down until refence - final posioning
	IF (STEP = 26) THEN
		myStatus = FC302_SEQ_Referencing
		Referencing					= TRUE
		RB[idx].Lift.RunForwards 	= FALSE
		RB[idx].Lift.RunReverse 	= EnableReference
		RB[idx].Lift.RunFreq		= 10  ;1Hz get exact location
		IF RB[idx].Lift.SeqIn.I_RefPosn THEN
			RB_Retain[idx].Lift.PosnRef = RB[idx].Lift.PosnAct
			RB[idx].Lift.SeqStep = 30
		ENDIF
	ENDIF

	;------------------
	;Auto tune Position
	;------------------

	EnableTune = NOT DisableDrive

	;Rail in correct position proximity - depending on which is required
	I_InPosition = FALSE
	IF (RB[idx].Lift.SeqIn.AutoTuneReceive = AlignReceive) THEN
		I_InPosition = RB[idx].Lift.SeqIn.I_RailOkReceive
	ELSE
		I_InPosition = RB[idx].Lift.SeqIn.I_RailOkRelease
	ENDIF

	;Check in rough position Release or Recieve Prox Made
	IF (STEP = 41) THEN
		myStatus = FC302_SEQ_AutoTune
		RB[idx].Lift.SeqOut.AutoTunePosn = RB[idx].Lift.SeqIn.AutoTunePosn ;Auto Tune Status back to sequence
		IF I_InPosition THEN
			RB[idx].Lift.SeqStep = 42
		ELSE
			;Do What?
		ENDIF
		IF (RB[idx].Lift.SeqIn.AutoTunePosn = 0) THEN
			RB[idx].Lift.SeqStep = 30 ;Cancel AutoTune
		ENDIF
	ENDIF

	;Move up until prox not made and store value
	IF (STEP = 42) THEN
		myStatus = FC302_SEQ_AutoTune
		RB[idx].Lift.RunForwards 	= EnableTune
		RB[idx].Lift.RunReverse 	= FALSE
		RB[idx].Lift.RunFreq		= 10
		IF NOT I_InPosition THEN
			AutoSavedTop			= RB[idx].Lift.PosnNow
			RB[idx].Lift.SeqStep 	= 43
		ENDIF
		IF (RB[idx].Lift.SeqIn.AutoTunePosn = 0) THEN
			RB[idx].Lift.SeqStep = 30 ;Cancel AutoTune
		ENDIF
	ENDIF

	;Move down until prox made
	IF (STEP = 43) THEN
		myStatus = FC302_SEQ_AutoTune
		RB[idx].Lift.RunForwards 	= FALSE
		RB[idx].Lift.RunReverse 	= EnableTune
		RB[idx].Lift.RunFreq		= 10
		IF I_InPosition THEN
			RB[idx].Lift.SeqStep 	= 44
		ENDIF
		IF (RB[idx].Lift.SeqIn.AutoTunePosn = 0) THEN
			RB[idx].Lift.SeqStep = 30 ;Cancel AutoTune
		ENDIF
	ENDIF

	;Move down until prox not made and calc position difference
	IF (STEP = 44) THEN
		myStatus = FC302_SEQ_AutoTune
		RB[idx].Lift.RunForwards 	= FALSE
		RB[idx].Lift.RunReverse 	= EnableTune
		RB[idx].Lift.RunFreq		= 10
		IF NOT I_InPosition THEN
			AutoSavedBottom			= RB[idx].Lift.PosnNow
			RB[idx].Lift.SeqStep 	= 45
		ENDIF
		IF (RB[idx].Lift.SeqIn.AutoTunePosn = 0) THEN
			RB[idx].Lift.SeqStep = 30 ;Cancel AutoTune
		ENDIF
	ENDIF

	;Store new position
	IF (STEP = 45) THEN

		myStatus = FC302_SEQ_AutoTune

		;Calculate position
		AutoPosnDiff = ((AutoSavedTop - AutoSavedBottom) / 2)
		AutoNewPosn  = (AutoSavedTop - AutoPosnDiff)

		RB_Posn[idx].Lift.Posn[RB[idx].Lift.SeqIn.AutoTunePosn] = AutoNewPosn

		RB[idx].Lift.SeqOut.AutoTunePosn = 0 ;Clear Auto Position
		RB[idx].Lift.SeqStep = 46

	ENDIF

	;Wait until RB sequence has cancelled auto position
	IF (STEP = 46) THEN
		IF (RB[idx].Lift.SeqIn.AutoTunePosn = 0) THEN
			RB[idx].Lift.SeqStep = 30
		ENDIF
	ENDIF

	;Read a parameter - not used at present
	IF ((STEP < 11) OR (STEP > 14)) AND (RB[idx].Lift.CAN.ModuleOk OR (RB[idx].Lift.CAN.NodeStatus = 3)) THEN

		IF ParameterEnable THEN

		//	D[85] = MonitorIdx

			MonitorSubIndex = 0
			IF (MonitorIdx = 1) THEN
				MonitorIndex 	= 1610 ;Motor Power
			ELSE IF (MonitorIdx = 2) THEN
				MonitorIndex 	= 1612 ;Motor Voltage
			ELSE IF (MonitorIdx = 3) THEN
				MonitorIndex 	= 1613 ;Motor Hz
			ELSE IF (MonitorIdx = 4) THEN
				MonitorIndex 	= 1614 ;Motor A
			ELSE IF (MonitorIdx = 5) THEN
				MonitorIndex 	= 1616 ;Motor Torque Nm
			ELSE IF (MonitorIdx = 6) THEN
				MonitorIndex 	= 1617 ;Motor RPM
			ELSE IF (MonitorIdx = 7) THEN
				MonitorIndex 	= 1634 ;Drive °C
			ELSE IF (MonitorIdx = 8) THEN
				MonitorIndex 	= 1502 ;Motor kWh
			ELSE IF (MonitorIdx = 9) THEN
				MonitorIndex 	= 1690 ;Alarm word
			ELSE IF (MonitorIdx = 10) THEN
				MonitorIndex 	= 1691 ;Alarm word 2
			ELSE IF (MonitorIdx = 11) THEN
				MonitorIndex 	= 1692 ;Warning word
			ELSE IF (MonitorIdx = 12) THEN
				MonitorIndex 	= 1693 ;Warning word 2
			ELSE
				MonitorIdx = 1
			ENDIF

			;Monitor caused CAN problems do not use!!
			;----------------------------------------
			;FC302_ReadParam_0.enable 	= TRUE
			;FC302_ReadParam_0.pDevice 	= ADR(sDevice)
			;FC302_ReadParam_0.node 		= node
			;FC302_ReadParam_0.index 	= MonitorIndex
			;FC302_ReadParam_0.subindex 	= MonitorSubIndex
			;FC302_ReadParam_0 FUB FC302_ReadParam()

			;IF (FC302_ReadParam_0.status = 0) THEN
			;	myRead 	= UINT(FC302_ReadParam_0.data)
			;ENDIF

			RB[idx].Lift.Motor.Value = INT(myRead)
			RB_Posn[idx].Lift.Monitor = INT(myRead)

		ENDIF

	ENDIF

	;Normal Operation
	IF (STEP = 30) THEN

		IF (mySlowWindow = 0) THEN
			mySlowWindow = 500 ;200 ;1000
		ENDIF
		IF (myDist = 0) THEN
			myDist = 250 ;200
		ENDIF

		RB[idx].Lift.SeqOut.RefComplete = TRUE

		;Power Save mode changed - re-calculate run speed
		IF PowerSave <> RB[idx].Lift.SeqIn.PowerSave THEN
			RB[idx].Lift.RunHz 	= 0
			PowerSave 			= RB[idx].Lift.SeqIn.PowerSave
		ENDIF

		;Calculate the required speed and stop distance with each run signal
		IF RB[idx].Lift.SeqIn.Run THEN
			IF (RB[idx].Lift.RunHz = 0) THEN
				;Required speed
				MotorNomHz 				= 50	;Motor nominal speed 50Hz
				RampTime 				= 10 	;1.0 sec - Read value in future?
				RampDist				= ((MotorNomHz * RB[idx].Lift.mmPerHz) * RampTime) ;Nominal Ramp Dist @ 50Hz
				DistRemain				= RB[idx].Lift.DistRemain
				RampFactor 				= (DistRemain / RampDist) ;eg 500mm Remain / 620mm (RampDist @ 50Hz) = 0.8
				RequiredHz				= UINT((MotorNomHz * RampFactor) * 10)
				MaxHz					= UINT((RB[idx].Lift.SeqIn.MaxSpeed / RB[idx].Lift.mmPerHz) * 10)
				;Restrict speed to value from sequence or 1000mm/sec (80.6 Hz)
				;IF (MaxHz > 806) THEN
				;	MaxHz = 806
				;ENDIF
				IF (MaxHz > 1209) THEN
					MaxHz = 1209
				ENDIF
				IF (RequiredHz > MaxHz) THEN
					RB[idx].Lift.RunHz 	= MaxHz
				ELSE
					RB[idx].Lift.RunHz 	= RequiredHz
				ENDIF
				;Stop Distance
				;RB[idx].Lift.StopDist 	= (((RB[idx].Lift.RunHz * RB[idx].Lift.SeqIn.RunSpeed) * RampTime) / 1000)
				StopFactor				= (REAL(RB[idx].Lift.RunHz) / (MotorNomHz * 10))
				RunSpeed				= (StopFactor * (RampDist / 10))
				RB[idx].Lift.StopDist	= UDINT((RunSpeed * StopFactor) / 0.2)
				SlowWindow 				= mySlowWindow ;1000 ;10tenths mm - try lower larger than CAN scan time
				StopDist				= RB[idx].Lift.StopDist + SlowWindow
			ENDIF

		ELSE
			RB[idx].Lift.RunHz = 0
		ENDIF

		;Position Required?
		IF (RB[idx].Lift.DistRemain > StopDist) THEN
			RB[idx].Lift.RunFreq 	= RB[idx].Lift.RunHz
		ELSE IF (RB[idx].Lift.DistRemain > myDist) THEN ;200) THEN 	;100 = 10mm
			RB[idx].Lift.RunFreq = 81 					;8.1Hz = 100mm/sec
		ELSE IF (RB[idx].Lift.DistRemain > 5) 	THEN 	;5 = 0.5mm
			RB[idx].Lift.RunFreq = 12					;1.2Hz, 0.8Hz = 10mm/sec
		ELSE
			RB[idx].Lift.RunFreq = 0
		ENDIF

		;Final Ramp Time
		IF (RB[idx].Lift.RunFreq = RB[idx].Lift.RunHz) THEN
			RB[idx].Lift.RampStart 	= 0
			RB[idx].Lift.RampTime 	= 0
		ELSE IF (RB[idx].Lift.RunFreq > 0) THEN
			IF (RB[idx].Lift.RampStart = 0) THEN
				RB[idx].Lift.RampStart = clock_ms()
			ENDIF
		ELSE IF (RB[idx].Lift.RunFreq = 0) THEN
			IF (RB[idx].Lift.RampTime = 0) THEN
				RB[idx].Lift.RampTime = (clock_ms() - TIME(RB[idx].Lift.RampStart))
			ENDIF
			;Store Max final ramp time
			IF (RB[idx].Lift.RampTime > RB[idx].Lift.RampMax) THEN
				RB[idx].Lift.RampMax = RB[idx].Lift.RampTime
			ENDIF
		ENDIF

		RB[idx].Lift.RunForwards 	= (RB[idx].Lift.SeqIn.Run AND (RB[idx].Lift.PosnNow < RB[idx].Lift.SeqIn.PosnReq))
		RB[idx].Lift.RunReverse 	= (RB[idx].Lift.SeqIn.Run AND (RB[idx].Lift.PosnNow > RB[idx].Lift.SeqIn.PosnReq))

		;Check Rail Alignment Switches
		IF RB[idx].Lift.SeqIn.Run THEN
			IF NOT AlignSwitchCheck THEN
				AlignSwitchCheck 	= TRUE
				ReleaseSwitchOk 	= FALSE
				ReceiveSwitchOk		= FALSE
			ENDIF
		ELSE
			AlignSwitchCheck = FALSE
		ENDIF

		;Switches have gone off during operation
		IF NOT RB[idx].Lift.SeqIn.I_RailOkRelease THEN
			ReleaseSwitchOk = TRUE
		ENDIF

		IF NOT RB[idx].Lift.SeqIn.I_RailOkReceive THEN
			ReceiveSwitchOk = TRUE
		ENDIF
		;------------------------------

		RailAligned = FALSE
		IF (RB[idx].Lift.SeqIn.RailAlign = AlignNone) THEN
			RailAligned	= TRUE
		ELSE IF (RB[idx].Lift.SeqIn.RailAlign = AlignReceive) AND RB[idx].Lift.SeqIn.I_RailOkReceive THEN
			RailAligned	= TRUE
		ELSE IF (RB[idx].Lift.SeqIn.RailAlign = AlignRelease) AND RB[idx].Lift.SeqIn.I_RailOkRelease THEN
			RailAligned	= TRUE
		ENDIF
		PosnValid					= (RB[idx].Lift.DistRemain <= 10) ;10=1mm
		AlignSwitchesOk				= (ReleaseSwitchOk AND ReceiveSwitchOk)
		RB[idx].Lift.SeqOut.PosnOk  = ((RB[idx].Lift.RunFreq = 0) AND PosnValid AND RailAligned AND AlignSwitchesOk)

		IF ((RB[idx].Lift.RunFreq = 0) AND PosnValid) THEN
			IF NOT RailAligned THEN
				myStatus = FC302_SEQ_RailNotAligned
			ELSE IF NOT ReleaseSwitchOk THEN
				myStatus = FC302_SEQ_ReleaseSwitchFault
			ELSE IF NOT ReceiveSwitchOk THEN
				myStatus = FC302_SEQ_ReceiveSwitchFault
			ENDIF
		ENDIF

		;Reference Check - CHeck position when moving down onto reference switch..

		;Travel limit reached go-to reference
		;IF NOT LimitsOk THEN
		;	RB[idx].Lift.SeqStep = 0
		;ENDIF

		;No reference position then go-to reference
		IF (RB_Retain[idx].Lift.PosnRef = 0) THEN
			RB[idx].Lift.SeqStep = 0
		ENDIF

		;Go to Manual Jog
		IF (RB[idx].Lift.SeqIn.JogForwards OR RB[idx].Lift.SeqIn.JogReverse) THEN
			JogHz				 = 100
			RB[idx].Lift.SeqStep = 32
		ENDIF

		;Auto fine tune required?
		IF (RB[idx].Lift.SeqIn.AutoTunePosn > 0) THEN
			RB[idx].Lift.SeqStep = 41
		ENDIF

		;Drive disable request or e-stop from sequence
		IF DisableDrive THEN
			RB[idx].Lift.SeqStep = 31
		ENDIF

	ELSE
		RB[idx].Lift.RunHz = 0
	ENDIF ;\Step 30

	;Drive Disabled - RB Sequence stops drive operation
	IF (STEP = 31) THEN
		RB[idx].Lift.SeqOut.RefComplete 	= TRUE
		RB[idx].Lift.SeqOut.DriveDisabled 	= DisableDrive
		IF NOT DisableDrive THEN
			RB[idx].Lift.SeqStep = 30
		ENDIF
	ELSE IF Referencing THEN
		RB[idx].Lift.SeqOut.DriveDisabled 	= DisableDrive
	ENDIF

	;RB Seq Do Reference Received
	IF (STEP <> 31) THEN
		IF RB[idx].Lift.SeqIn.DoRef THEN
			RB[idx].Lift.SeqIn.DoRef 	= FALSE
			IF (RB[idx].Lift.CAN.NodeStatus = 261) THEN
				RB[idx].Lift.SeqStep = 21
			ELSE
				RB[idx].Lift.SeqStep = 0
			ENDIF
		ENDIF
	ENDIF

	;Enable reset of drive when in error - trip lock and drive not ready etc..
	IF ((STEP = 31) AND NOT RB[idx].Lift.SeqIn.DisableDrive) THEN
		IF RB[idx].Lift.SeqIn.DoRef THEN
			RB[idx].Lift.SeqIn.DoRef 	= FALSE
			RB[idx].Lift.SeqStep 		= 0
		ENDIF
	ENDIF

	;Jog mode - 1 second slow before accelleration
	TmrJog.IN = (STEP = 32)
	TmrJog.PT = 100
	TmrJog FUB TON_10ms()
	IF (STEP = 32) THEN
		myStatus = FC302_SEQ_Jog
		Referencing					= TRUE
		RB[idx].Lift.RunForwards 	= RB[idx].Lift.SeqIn.JogForwards
		RB[idx].Lift.RunReverse 	= RB[idx].Lift.SeqIn.JogReverse
		RB[idx].Lift.RunFreq		= (JogHz / 10)
		IF (TmrJog.Q AND (JogHz < 1600)) THEN ;160 (1600 / 10) around 200mm/sec
			JogHz = JogHz + 1 ;Acc by 0.1 Hz / Scan 81 = 8.1Hz = 100mm/sec
		ENDIF
		IF (NOT RB[idx].Lift.SeqIn.JogForwards AND NOT RB[idx].Lift.SeqIn.JogReverse) THEN
			RB[idx].Lift.SeqStep = 30
		ENDIF
	ENDIF

	EnableForwards 	= (RB[idx].Lift.RunForwards AND RB[idx].Lift.SeqIn.I_ForwardLimitOk)
	EnableReverse	= (RB[idx].Lift.RunReverse  AND RB[idx].Lift.SeqIn.I_ReverseLimitOk)

	EnableDrive 	= (NOT DisableDrive AND (EnableForwards OR EnableReverse) AND (RB[idx].Lift.RunFreq > 0))

	QuickStop		= (RB[idx].Lift.SeqIn.EStop OR (NOT Referencing AND (NOT RB[idx].Lift.SeqIn.I_ForwardLimitOk OR NOT RB[idx].Lift.SeqIn.I_ReverseLimitOk)))
	;QuickStop		= RB[idx].Lift.SeqIn.EStop

	;Estop
	;Drive ready from status word and bus control

	;Give current position to RB sequence
	RB[idx].Lift.SeqOut.PosnNow = INT(RB[idx].Lift.PosnNow / 10)

	;Drive Control Word
	IF RB[idx].Lift.CAN.ModuleOk THEN
		IF EnableDrive AND NOT QuickStop THEN
			RB[idx].Lift.CTW.DC_Brake		= TRUE
			RB[idx].Lift.CTW.Coasting		= TRUE
			RB[idx].Lift.CTW.QuickStop		= (RB[idx].Lift.RunFreq > 0)
			RB[idx].Lift.CTW.HoldOutputFreq	= TRUE
			RB[idx].Lift.CTW.RampStopStart	= TRUE
			RB[idx].Lift.CTW.ResetTrip		= FALSE
			RB[idx].Lift.CTW.DataValid		= TRUE
			RB[idx].Lift.CTW.Reverse		= EnableForwards  	;Due to mechanical arrangement Reverse is Up/Forwards
			RB[idx].Lift.CAN.TargetVelocity	= UINT(($4000 / 1000) * RB[idx].Lift.RunFreq)
		ELSE
			RB[idx].Lift.CTW.DC_Brake		= FALSE//TRUE
			RB[idx].Lift.CTW.Coasting		= TRUE
			RB[idx].Lift.CTW.QuickStop		= FALSE// NOT QuickStop ;0 = QuickStop
			RB[idx].Lift.CTW.HoldOutputFreq	= FALSE//TRUE
			RB[idx].Lift.CTW.RampStopStart	= FALSE
			RB[idx].Lift.CTW.ResetTrip		= FALSE
			RB[idx].Lift.CTW.DataValid		= TRUE
			RB[idx].Lift.CTW.Reverse		= FALSE
			RB[idx].Lift.CAN.TargetVelocity	= $0000
		ENDIF
	ENDIF

	;Write control word to drive
	FC302_WriteCTW_0.CTW = RB[idx].Lift.CTW
	FC302_WriteCTW_0 FUB FC302_WriteCTW()
	RB[idx].Lift.CAN.ControlWord = FC302_WriteCTW_0.ControlWord

	;Scan time calculation
	IF NOT RB[idx].Lift.Scan.StartTrig AND NOT RB[idx].Lift.Scan.EndTrig THEN
		IF RB[idx].Lift.CTW.RampStopStart THEN
			RB[idx].Lift.Scan.Start 	= clock_ms()
			RB[idx].Lift.Scan.StartTrig = TRUE
		ENDIF
	ELSE IF RB[idx].Lift.Scan.StartTrig AND NOT RB[idx].Lift.Scan.EndTrig THEN
		IF RB[idx].Lift.STW.InOperation THEN
			RB[idx].Lift.Scan.End 		= clock_ms()
			RB[idx].Lift.Scan.EndTrig	= TRUE

			RB[idx].Lift.Scan.LastScan = UINT(RB[idx].Lift.Scan.End - RB[idx].Lift.Scan.Start)
			IF ((RB[idx].Lift.Scan.LastScan < RB[idx].Lift.Scan.MinScan) OR (RB[idx].Lift.Scan.MinScan = 0)) THEN
				RB[idx].Lift.Scan.MinScan = RB[idx].Lift.Scan.LastScan
			ENDIF
			IF (RB[idx].Lift.Scan.LastScan > RB[idx].Lift.Scan.MaxScan) THEN
				RB[idx].Lift.Scan.MaxScan = RB[idx].Lift.Scan.LastScan
			ENDIF
		ENDIF
	ELSE IF NOT RB[idx].Lift.CTW.RampStopStart AND NOT RB[idx].Lift.STW.InOperation THEN
		RB[idx].Lift.Scan.StartTrig = FALSE
		RB[idx].Lift.Scan.EndTrig 	= FALSE
	ENDIF

	;Status Word Warnings and Alarms
	IF RB[idx].Lift.STW.Trip THEN
		myStatus = FC302_STW_Trip
	ELSE IF RB[idx].Lift.STW.Error THEN
		myStatus = FC302_STW_Error
	ELSE IF RB[idx].Lift.STW.TripLock THEN
		myStatus = FC302_STW_TripLock
	ELSE IF RB[idx].Lift.STW.Warning THEN
		myStatus = FC302_STW_Warning
	ELSE IF RB[idx].Lift.STW.DriveOverTemp THEN
		myStatus = FC302_STW_DriveOverTemp
	ELSE IF RB[idx].Lift.STW.DriveVoltageFault THEN
		myStatus = FC302_STW_DriveVoltageFault
	ELSE IF RB[idx].Lift.STW.DriveTorqueLimit THEN
		myStatus = FC302_STW_DriveTorqueLimit
	ELSE IF RB[idx].Lift.STW.ThermalTimerLimit THEN
		myStatus = FC302_STW_ThermalTimeLimit
	ENDIF

	RB[idx].Lift.SeqOut.Status = myStatus

	;I/O Status to TrackView
	;-----------------------

	;Lift
	RB_Posn[idx].Lift.IOStatus  = 0 ;Clear
	IF RB[idx].Lift.SeqIn.I_RefPosn THEN
		RB_Posn[idx].Lift.IOStatus = BIT_SET(RB_Posn[idx].Lift.IOStatus, 0)
	ENDIF
	IF NOT RB[idx].Lift.SeqIn.I_ForwardLimitOk THEN
		RB_Posn[idx].Lift.IOStatus = BIT_SET(RB_Posn[idx].Lift.IOStatus, 1)
	ENDIF
	IF NOT RB[idx].Lift.SeqIn.I_ReverseLimitOk THEN
		RB_Posn[idx].Lift.IOStatus = BIT_SET(RB_Posn[idx].Lift.IOStatus, 2)
	ENDIF
	IF RB[idx].Lift.SeqIn.I_RailOkRelease THEN
		RB_Posn[idx].Lift.IOStatus = BIT_SET(RB_Posn[idx].Lift.IOStatus, 3)
	ENDIF
	IF RB[idx].Lift.SeqIn.I_RailOkReceive THEN
		RB_Posn[idx].Lift.IOStatus = BIT_SET(RB_Posn[idx].Lift.IOStatus, 4)
	ENDIF

END_PROGRAM
```

### Program Logical/SAFETY_ZONES (IEC, version 1.00.1) - SAFETY_ZONES

#### SAFETY_ZONES.st
```iecst
(********************************************************************
 * Program: safety_zones
 * File: safety_zones.st
 ********************************************************************)
PROGRAM _CYCLIC
	r1.safety_zone := SafetyZone[1].HaltSys;
	r2.safety_zone := SafetyZone[1].HaltSys;
	r3.safety_zone := SafetyZone[1].HaltSys;
	r4.safety_zone := SafetyZone[1].HaltSys;
	r5.safety_zone := SafetyZone[1].HaltSys;
	r6.safety_zone := SafetyZone[1].HaltSys;
	r7.safety_zone := SafetyZone[1].HaltSys;
	r8.safety_zone := SafetyZone[1].HaltSys;
	r9.safety_zone := SafetyZone[1].HaltSys;
	r10.safety_zone := SafetyZone[1].HaltSys;
	r11.safety_zone := SafetyZone[1].HaltSys;
	r12.safety_zone := SafetyZone[1].HaltSys;
	r13.safety_zone := SafetyZone[1].HaltSys;
	r14.safety_zone := SafetyZone[1].HaltSys;
	r15.safety_zone := SafetyZone[1].HaltSys;
	r16.safety_zone := SafetyZone[1].HaltSys;
	r17.safety_zone := SafetyZone[1].HaltSys;
	r18.safety_zone := SafetyZone[1].HaltSys;
	r19.safety_zone := SafetyZone[1].HaltSys;
	r20.safety_zone := SafetyZone[1].HaltSys;
	r21.safety_zone := SafetyZone[1].HaltSys;
	r22.safety_zone := SafetyZone[1].HaltSys;
	r23.safety_zone := SafetyZone[1].HaltSys;
	r24.safety_zone := SafetyZone[1].HaltSys;
	r25.safety_zone := SafetyZone[1].HaltSys;
	r26.safety_zone := SafetyZone[1].HaltSys;
	r27.safety_zone := SafetyZone[1].HaltSys;
	r28.safety_zone := SafetyZone[1].HaltSys;
	r29.safety_zone := SafetyZone[1].HaltSys;
	r30.safety_zone := SafetyZone[1].HaltSys;
	r31.safety_zone := SafetyZone[1].HaltSys;
	r32.safety_zone := SafetyZone[1].HaltSys;
	r33.safety_zone := SafetyZone[1].HaltSys;
	r34.safety_zone := SafetyZone[1].HaltSys;
	r35.safety_zone := SafetyZone[1].HaltSys;
	r36.safety_zone := SafetyZone[1].HaltSys;
	r37.safety_zone := SafetyZone[1].HaltSys;
	r38.safety_zone := SafetyZone[1].HaltSys;
	r39.safety_zone := SafetyZone[1].HaltSys;
	r40.safety_zone := SafetyZone[1].HaltSys;
	r41.safety_zone := SafetyZone[1].HaltSys;
	r42.safety_zone := SafetyZone[1].HaltSys;
	r43.safety_zone := SafetyZone[1].HaltSys;
	r44.safety_zone := SafetyZone[1].HaltSys;
	r45.safety_zone := SafetyZone[1].HaltSys;
	r46.safety_zone := SafetyZone[1].HaltSys;
	r47.safety_zone := SafetyZone[1].HaltSys;
	r48.safety_zone := SafetyZone[1].HaltSys;
	r49.safety_zone := SafetyZone[1].HaltSys;
	r50.safety_zone := SafetyZone[1].HaltSys;
	r51.safety_zone := SafetyZone[1].HaltSys;
	r52.safety_zone := SafetyZone[1].HaltSys;
	r53.safety_zone := SafetyZone[1].HaltSys;
	r54.safety_zone := SafetyZone[1].HaltSys;
	r55.safety_zone := SafetyZone[1].HaltSys;
	r56.safety_zone := SafetyZone[1].HaltSys;
	r57.safety_zone := SafetyZone[1].HaltSys;
	r58.safety_zone := SafetyZone[1].HaltSys;
	r59.safety_zone := SafetyZone[1].HaltSys;
	r60.safety_zone := SafetyZone[1].HaltSys;
	r61.safety_zone := SafetyZone[1].HaltSys;
	r62.safety_zone := SafetyZone[1].HaltSys;
	r63.safety_zone := SafetyZone[1].HaltSys;
	r64.safety_zone := SafetyZone[1].HaltSys;
	r65.safety_zone := SafetyZone[1].HaltSys;
	r66.safety_zone := SafetyZone[1].HaltSys;
	r67.safety_zone := SafetyZone[1].HaltSys;
	r68.safety_zone := SafetyZone[1].HaltSys;
	r69.safety_zone := SafetyZone[1].HaltSys;
	r70.safety_zone := SafetyZone[1].HaltSys;
	r71.safety_zone := SafetyZone[1].HaltSys;
	r72.safety_zone := SafetyZone[1].HaltSys;
	r73.safety_zone := SafetyZone[1].HaltSys;
	r74.safety_zone := SafetyZone[1].HaltSys;
END_PROGRAM
```

### Program Logical/BELT_TO_TRANSFER (IEC, version 1.00.1) - BELT_TO_TRANSFER

#### BELT_TO_TRANSFER.st
```iecst
(********************************************************************
 * Program: belt_to_transfer
 * File: belt_to_transfer.st
 ********************************************************************)
PROGRAM _CYCLIC

END_PROGRAM
```

### Program Logical/CONVEYOR_MAP (IEC, version 1.00.1) - CONVEYOR_MAP

#### CONVEYOR_MAP.st
```iecst
(********************************************************************
 * Program: conveyor_map
 * File: conveyor_map.st
 ********************************************************************)
PROGRAM _CYCLIC

END_PROGRAM
```

### Package Logical/COMMUNICATION - COMMUNICATION

### Communication.var
```iecst
(*Comm Config*)
VAR CONSTANT
  UDP_COMM_PORT : UINT := 4004;
  TCP_COMM_PORT : UINT := 12005;
END_VAR
(*Data sizes*)
VAR CONSTANT
  EVUE_COMM_BUFFER_SIZE : UINT := 20000; (*Size of data array for the memory map*)
  TCP_SEND_BUFFER_SIZE : UINT := 1000; (**Size of the send buffer for responses*)
  TCP_RECV_BUFFER_SIZE : UINT := 20000; (**Size of the recieve buffer*)
  UDP_SEND_PACKET_SIZE : UINT := 4000; (**Size of the packet to send*)
END_VAR
(***********UDP Comm Config************)
VAR CONSTANT
  LIVE_DATA_MAX_CONNECTIONS : USINT := 5; (**Maximum number of UDP Connections*)
  LIVE_DATA_MAX_POOL_SIZE : USINT := 10; (**Maximum number of data transmissions on 1 connection*)
END_VAR
(**)
(*DATA TYPE DEFINITIONS*)
VAR CONSTANT
  LIVE_DATA_TYPE_EVUE_UDP_COMM_1 : UINT := 1;
  LIVE_DATA_TYPE_EVUE_UDP_COMM_2 : UINT := 2;
  LIVE_DATA_TYPE_EVUE_UDP_COMM_3 : UINT := 3;
  LIVE_DATA_TYPE_EVUE_UDP_COMM_4 : UINT := 4;
  LIVE_DATA_TYPE_EVUE_UDP_COMM_5 : UINT := 5;
  LIVE_DATA_TYPE_RAIL_MESSAGES : UINT := 1001;
  LIVE_DATA_TYPE_SLING_INPUT_STATE : UINT := 3001;
END_VAR
(*DATA TYPE DEFINITIONS*)
VAR
        CommArray : ARRAY[0..EVUE_COMM_BUFFER_SIZE] OF UDINT; (**Global Array of pointers of comm vars*)
END_VAR
```

### Communication.typ
```iecst
(*USINT s sent in TCP as 2 bytes if it is not followed by another USINT ignore the upper*)

TYPE
  LiveData_RequestPool_typ : 	STRUCT
    AddToPool : UINT; (**Request to Add a Packet type to the request Pool*)
    RemoveFromPool : UINT; (**Request to Remove a Packet type from the pool*)
    PoolList : ARRAY[1..LIVE_DATA_MAX_POOL_SIZE]OF UINT; (**Pool List - (Data packets are polled through)*)
    PoolListSize : USINT; (**Size of the current Pool List*)
    Pointer : USINT; (**Pointer to active Packet*)
  END_STRUCT;
  LiveData_Tview_typ : 	STRUCT  (*Type 2 - Trackview data*)
    Header : LiveDataHeader_typ;
    HeaderCustom : ARRAY[0..99]OF USINT; (*Extra header information so Live DATA API can decode*)
    data : ARRAY[0..4]OF BOOL; (**To be built custom*)
  END_STRUCT;
END_TYPE

(*Data Frame ABB i s type 4 -- Defined in ABB Package*)
(*HEADER TYPE*)

TYPE
  LiveDataHeader_typ : 	STRUCT  (**Must be first part of all Data Frames*)
    Type : UINT; (*Byte 1*)
    HeaderSize : UINT; (*Byte 2 & 3*)
    Checksum : UDINT; (*Bytes 4 -7*)
  END_STRUCT;
  LiveDataHeaderCustom_typ : 	STRUCT  (**Standard Header with customer area*)
    Type : UINT; (*Byte 1*)
    HeaderSize : UINT; (*Byte 2 & 3*)
    Checksum : UDINT; (*Bytes 4 -7*)
    Custom : UINT; (*Bytes 8-9*)
  END_STRUCT;
END_TYPE

(*Insert your comment here.*)

TYPE
  LiveDataConnection_typ : 	STRUCT
    State : LiveDataConnectionState_enum; (**State of the connection*)
    RequestPool : LiveData_RequestPool_typ; (**Structure to manage to list of requested data types*)
    Config : LiveDataConnectionConfig_typ;
    Functions : LiveDataConnectionFunctions_typ;
    Error : UINT;
  END_STRUCT;
  LiveDataConnectionState_enum :
    (
    LIVE_DATA_INIT := 0,
    LIVE_DATA_WAIT := 10,
    LIVE_DATA_OPEN_CONNECTION := 20,
    LIVE_DATA_SETUP_CONNECTION_TOS := 30,
    LIVE_DATA_SETUP_CONNECTION_TTL := 31,
    LIVE_DATA_CONNECT := 40,
    LIVE_DATA_BUILD_DATA := 50,
    LIVE_DATA_SEND_DATA := 60,
    LIVE_DATA_CHECK_REQUESTPOOL := 70,
    LIVE_DATA_DISCONNECT := 80,
    LIVE_DATA_CLOSE_CONNECTION := 90,
    LIVE_DATA_ERROR := 200,
    LIVE_DATA_GET_IDENT_MAX := 210, (**Debugging functions*)
    LIVE_DATA_GET_IDENT_LIST := 220 (**Debugging functions*)
    );
  LiveDataConnectionFunctions_typ : 	STRUCT
    Open : UdpOpen;
    Ioctl : UdpIoctl;
    Connect : UdpConnect;
    Send : UdpSend;
    Disconnect : UdpDisconnect;
    Close : UdpClose;
  END_STRUCT;
  LiveDataConnectionConfig_typ : 	STRUCT
    ServerIP : STRING[16]; (**IP Address of Server*)
    ServerPort : UINT; (**Server connection Port*)
    Type : LiveDataConnectionConfig_enum;
    TTL : UDINT := 30; (*Time To Live MAx 255*)
    TOS : UDINT := 4;
  END_STRUCT;
  LiveDataConnectionConfig_enum :
    (
    LIVE_DATA_CONFIG_DYNAMIC_SERVER := 0, (*Idle connection listen on http server to start a connection*)
    LIVE_DATA_CONFIG_STATIC := 1, (*The IP and request are fixed and will be manually configured*)
    LIVE_DATA_CONFIG_DYNAMIC_CLIENT := 2 (*Use a Get request to load the Server Data and any required connections*)
    );
END_TYPE
```

### Library Logical/COMMUNICATION/MbusTCP (ANSIC, version 1.39.0)
Depends on: astcp, asstring, standard, AsARCfg, sys_lib

#### MbusTCP.typ
```iecst
TYPE
	modbus_slave_cfg_typ : 	STRUCT
		p_discrete_inputs : ARRAY[0..99]OF UDINT;
		p_coils : ARRAY[0..99]OF UDINT;
		p_input_registers : ARRAY[0..99]OF UDINT;
		p_holding_registers : ARRAY[0..20000]OF UDINT;
	END_STRUCT;
	master_info_typ : 	STRUCT
		ident : UDINT;
		port : UINT;
		ip_addr : ARRAY[0..17]OF USINT; (*Client IP address*)
		timeout_timer : TON; (*Timer to determine when connection times out*)
		disconnect : BOOL; (*Flag to disconnect this client if it times out.*)
	END_STRUCT;
	receive_buff_typ : 	STRUCT  (*Receive data buffer*)
		byte : ARRAY[0..32000]OF USINT; (*Received data*)
	END_STRUCT;
	modbus_master_action_enable_typ : 	STRUCT
		cyclic : BOOL;
		single : BOOL;
	END_STRUCT;
	modbus_master_action_param_typ : 	STRUCT
		unit : USINT;
		type : USINT;
		start_addr : UINT;
		quantity : UINT;
		p_pv : UDINT;
		timer : UDINT;
	END_STRUCT;
	modbus_master_cfg_typ : 	STRUCT
		action_enable : ARRAY[0..19]OF modbus_master_action_enable_typ;
		action_param : ARRAY[0..19]OF modbus_master_action_param_typ;
	END_STRUCT;
	modbus_master_internal_typ : 	STRUCT  (*Internal master variables*)
		step : UINT; (*Internal state in a state machine*)
		tcp_open : TcpOpen; (*TcpOpen FUB from AsTCP*)
		tcp_ioctl : TcpIoctl; (*TcpIoctl FUB from AsTCP*)
		tcp_client : TcpClient; (*TcpClient FUB from AsTCP*)
		tcp_send : TcpSend; (*TcpSend FUB from AsTCP*)
		tcp_receive : TcpRecv; (*TcpRecv FUB from AsTCP*)
		tcp_close : TcpClose; (*TcpClose FUB from AsTCP*)
		tcp_ip : CfgGetIPAddr;
		linger_opt : tcpLINGER_typ; (*TcpIoctl linger options*)
		last_req : USINT; (*Last request*)
		receive_timer : UDINT; (*Receive timer*)
		send_timer : ARRAY[0..19]OF UDINT; (*Send timer*)
		send_buff : ARRAY[0..500]OF USINT; (*Send buffer*)
		receive_buff : ARRAY[0..500]OF USINT; (*Receive buffer*)
		transaction_id : UINT; (*Transaction ID*)
		wrong_message : UDINT; (*Wrong message counter*)
	END_STRUCT;
	modbus_log_typ : 	STRUCT  (*Log of data for the ModbusTCP FUBs*)
		data_lines : UINT; (*Number of character lines in the log*)
		pData : UDINT; (*Pointer to the log buffer*)
	END_STRUCT;
	modbus_slave_internal_typ : 	STRUCT  (*Internal slave variables*)
		step : UINT; (*Internal state in a state machine*)
		substep : UINT; (*Internal substate in a state machine*)
		i : USINT; (*Loop counter*)
		master_nr : USINT; (*Client ID*)
		master_last : USINT;
		master_info : ARRAY[0..10]OF master_info_typ; (*Client info*)
		master_addr : ARRAY[0..17]OF USINT; (*Client IP address*)
		tcp_open : TcpOpen; (*TcpOpen FUB from AsTCP*)
		tcp_ioctl : TcpIoctl; (*TcpIoctl FUB from AsTCP*)
		tcp_server : TcpServer; (*TcpServer FUB from AsTCP*)
		tcp_send : TcpSend; (*TcpSend FUB from AsTCP*)
		tcp_receive : ARRAY[0..10]OF TcpRecv; (*TcpRecv FUB from AsTCP*)
		tcp_close : TcpClose; (*TcpClose FUB from AsTCP*)
		tcp_ip : CfgGetIPAddr;
		linger_opt : tcpLINGER_typ; (*TcpIoctl linger options*)
		send_buff : ARRAY[0..32000]OF USINT; (*Send buffer*)
		send_byte : UINT;
		receive_buff : ARRAY[0..10]OF receive_buff_typ; (*Receive buffers for clients*)
		open_connections : ARRAY[0..254]OF UDINT; (*Open Connections*)
		connection_pointer : UINT;
	END_STRUCT;
END_TYPE
```

#### MBmaster.c - Master
```c
/********************************************************************
 * COPYRIGHT --
 ********************************************************************
 * Library: MbusTCP
 * Author: strickers
 * Created: October 29, 2009
 *******************************************************************/
#include <MBdeclarations.h>

/* ------------------------------------------------------------------------------------------------- */
/* Local functions */
/* ------------------------------------------------------------------------------------------------- */
UINT create_request_to_slave	(modbus_master_cfg_typ* config, USINT req_nr, USINT* send_buff, UINT size_buf, UINT transaction_id, modbus_log_typ LOGBOOK);
UINT analyze_answer_from_slave	(modbus_master_cfg_typ*	config,	USINT req_nr, USINT* receive_buff, UINT	transaction_id, modbus_log_typ LOGBOOK);

/* ------------------------------------------------------------------------------------------------- */
/* Master function block */
/* ------------------------------------------------------------------------------------------------- */
void MBmaster(MBmaster_typ* inst)
{
	USINT	x;
	USINT	receive_status;

	/* Increase cycle timers when connected */
	if(inst->internal.step > WAIT_CONNECTION)
	{
		/* Make sure cycle time has a value */
		if((inst->cycle_time == 0) && (inst->internal.step != ERROR))
		{
			NewLogEntry("ERR: Cyclic time is 0", inst->log);
			inst->status 		= ERROR_CYCLIC_ZERO;
			inst->internal.step = ERROR;
		}
		else
		{
			for(x=0;x<sizeof((*(inst->p_cfg)).action_param)/sizeof((*(inst->p_cfg)).action_param[0]);x++)
				inst->internal.send_timer[x] += inst->cycle_time;
		}
	}
	switch(inst->internal.step)
	{
		/* ------------------------------------------------------------------------------------------ */
		/* Assign buffers and port */
		case INIT:
			inst->internal.tcp_send.pData 		= (UDINT)inst->internal.send_buff;
			inst->internal.tcp_receive.pData	= (UDINT)inst->internal.receive_buff;
			inst->internal.tcp_receive.datamax	= sizeof(inst->internal.receive_buff);
			if(inst->port == 0) inst->port = MODBUS_TCP_PORT;
			inst->internal.step = DISABLE;
		/* ------------------------------------------------------------------------------------------ */
		/* Wait for function block enable */
		case DISABLE:
			if(inst->enable)
			{
				inst->internal.step = GET_IP;
				NewLogEntry("Validating own ip...", inst->log);
			}
		break;
		/* ------------------------------------------------------------------------------------------ */
		/* Read own IP address */
		case GET_IP:
			if(inst->enable)
			{
				inst->internal.tcp_ip.enable 	= 1;
				inst->internal.tcp_ip.pDevice 	= (UDINT)inst->device;
				inst->internal.tcp_ip.pIPAddr 	= (UDINT)inst->my_ip;
				inst->internal.tcp_ip.Len 		= 18;
				CfgGetIPAddr(&inst->internal.tcp_ip);
				inst->status = inst->internal.tcp_ip.status;
				/* -------------------------------------------------------------------------------------- */
				/* Success  */
				if (inst->internal.tcp_ip.status == 0)
				{
					if(strcmp(inst->my_ip, "0.0.0.0") == 0) break;
					inst->internal.step = OPEN_PORT;
				}
				else if(inst->internal.tcp_ip.status == cfgERR_DEVICE_NOT_EXIST)
				{
					NewLogEntry("ERR: Invalid ethernet device", inst->log);
					inst->status 		= ERROR_DEVICE_ERR;
					inst->internal.step = ERROR;
				}
				else if(inst->internal.tcp_ip.status != BUSY) inst->internal.step = ERROR;
			}
			else inst->internal.step = CLOSE_PORT;
		break;
		/* ------------------------------------------------------------------------------------------ */
		/* Open ethernet port */
		case OPEN_PORT:
			if(inst->enable)
			{
				inst->internal.tcp_open.options = tcpOPT_REUSEADDR;
				inst->internal.tcp_open.enable 	= 1;
				TcpOpen(&inst->internal.tcp_open);
				/* -------------------------------------------------------------------------------------- */
				/* Success  */
				if (inst->internal.tcp_open.status == 0)
				{
					NewLogEntry("Open port successful", inst->log);
					inst->internal.tcp_client.enable	= 1;
					inst->internal.tcp_client.ident		= inst->internal.tcp_open.ident;
					inst->internal.tcp_client.pServer	= (UDINT)inst->slave_ip_addr;
					inst->internal.tcp_client.portserv	= inst->port;
					inst->internal.tcp_send.ident		= inst->internal.tcp_open.ident;
					inst->internal.tcp_receive.ident	= inst->internal.tcp_open.ident;
					NewLogEntry("Trying to connect...", inst->log);
					inst->internal.step = WAIT_CONNECTION;
				}
				else if(inst->internal.tcp_open.status != BUSY) inst->internal.step = ERROR;
				inst->status = inst->internal.tcp_open.status;
			}
			else inst->status = 65534;
		break;
		/* ------------------------------------------------------------------------------------------ */
		/* Open ethernet port */
		case WAIT_CONNECTION:
			if(inst->enable)
			{
				inst->internal.tcp_client.enable = 1;
				TcpClient(&inst->internal.tcp_client);
				inst->status = inst->internal.tcp_client.status;
				/* ---------------------------------------------------------------------------------- */
				/* Success */
				if(inst->internal.tcp_client.status == 0)
				{
					NewLogEntry("Connected", inst->log);
					inst->internal.step = CREATE_REQUEST;
				}
				else if(inst->internal.tcp_client.status == tcpERR_INVALID)
				{
					NewLogEntry("ERR: Cant find slave", inst->log);
					inst->status = ERROR_TIMEOUT_CONNECT;
					inst->internal.step = CLOSE_PORT;
				}
				else if(inst->internal.tcp_client.status != BUSY)
				{
					NewLogEntry("ERR: Could not establish connection", inst->log);
					inst->status = ERROR_TIMEOUT_CONNECT;
					inst->internal.step = ERROR;
				}
			}
			else inst->internal.step = CLOSE_PORT;
		break;
		/* ------------------------------------------------------------------------------------------ */
		/* Create new requests  */
		case CREATE_REQUEST:
			if(inst->enable)
			{
				UINT tmp_req = inst->internal.last_req;
				/* ---------------------------------------------------------------------------------- */
				/* Find next request */
				do
				{
					/* ---------------------------------------------------------------------------------- */
					/* Switch to next action, roll over */
					inst->internal.last_req++;
					if(((*(inst->p_cfg)).action_param[inst->internal.last_req].p_pv == 0) || (inst->internal.last_req >= sizeof((*(inst->p_cfg)).action_param)/sizeof((*(inst->p_cfg)).action_param[0]))) inst->internal.last_req=0;
					/* ---------------------------------------------------------------------------------- */
					/* Execute action when set to single or timer is expired */
					if (((*(inst->p_cfg)).action_enable[inst->internal.last_req].single) ||
						((inst->internal.send_timer[inst->internal.last_req] >= (*(inst->p_cfg)).action_param[inst->internal.last_req].timer) && ((*(inst->p_cfg)).action_enable[inst->internal.last_req].cyclic)))
					{
						if(((*(inst->p_cfg)).action_param[inst->internal.last_req].p_pv) != 0)
						{
							inst->internal.step = SEND_REQUEST;
							inst->internal.transaction_id++;
							inst->internal.tcp_send.datalen = create_request_to_slave((modbus_master_cfg_typ*)(inst->p_cfg), inst->internal.last_req, inst->internal.send_buff, sizeof(inst->internal.send_buff), inst->internal.transaction_id, inst->log);
							inst->internal.send_timer[inst->internal.last_req] = 0;
						}
						else /* Variable address is empty */
						{
						NewLogEntry("ERR: Empty variable ADR", inst->log);
						inst->status 		= ERROR_ADR_EMPTY;
						inst->internal.step = ERROR;
						}
						break;
					}
					if(inst->internal.last_req == tmp_req) break;
				}
				while(1);
			}
			else inst->internal.step = CLOSE_PORT;
		break;
		/* ------------------------------------------------------------------------------------------ */
		/* Create new requests */
		case SEND_REQUEST:
			if(inst->enable)
			{
				inst->internal.tcp_send.enable = 1;
				TcpSend(&inst->internal.tcp_send);
				/* ---------------------------------------------------------------------------------- */
				/* Success */
				if(inst->internal.tcp_send.status == 0)
				{
					inst->internal.receive_timer = 0;
					inst->internal.step = WAIT_ANSWER;
				}
				else if(((inst->internal.tcp_send.status != BUSY) 				&&
					     (inst->internal.tcp_send.status != tcpERR_WOULDBLOCK)	&&
					     (inst->internal.tcp_send.status != tcpERR_SENTLEN))    ||
						 (inst->internal.tcp_send.status == tcpERR_NOT_CONNECTED))	inst->internal.step = CLOSE_PORT;
			}
			else inst->internal.step = CLOSE_PORT;
			inst->status = inst->internal.tcp_send.status;
		break;
		/* ------------------------------------------------------------------------------------------ */
		/* Wait for answer */
		case WAIT_ANSWER:
			if(inst->enable)
			{
				inst->internal.tcp_receive.enable = 1;
				TcpRecv(&inst->internal.tcp_receive);
				/* ---------------------------------------------------------------------------------- */
				/* Success */
				if(inst->internal.tcp_receive.status == 0)
				{
					if(inst->internal.tcp_receive.recvlen != 0)
					{
						if((inst->internal.tcp_receive.recvlen > 8) && (inst->internal.tcp_receive.recvlen < sizeof(inst->internal.receive_buff)))
						{
							receive_status = analyze_answer_from_slave((modbus_master_cfg_typ*)(inst->p_cfg), inst->internal.last_req, inst->internal.receive_buff, inst->internal.transaction_id, inst->log);
							if(receive_status) inst->last_error = ERROR_BAD_SLAVE_DATA;
						}
						else if(inst->internal.tcp_receive.recvlen >= sizeof(inst->internal.receive_buff))
						{
							NewLogEntry("ERR: Data received too long", inst->log);
							receive_status = 1;
							inst->last_error = ERROR_SLAVE_DATA_TOO_LONG;
						}
						else
						{
							NewLogEntry("ERR: Data received too short", inst->log);
							receive_status = 1;
							inst->last_error = ERROR_SLAVE_DATA_TOO_SHORT;
						}
						if(receive_status) 	inst->internal.wrong_message ++;
						(*(inst->p_cfg)).action_enable[inst->internal.last_req].single = 0;
						inst->internal.step = CREATE_REQUEST;
					}
					else inst->internal.step = CLOSE_PORT;
				}
				else if((inst->internal.tcp_receive.status != BUSY) &&
					    (inst->internal.tcp_receive.status != tcpERR_NO_DATA)) inst->internal.step = CLOSE_PORT;
				/* ---------------------------------------------------------------------------------- */
				/* See if request timed out */
				inst->internal.receive_timer += inst->cycle_time;
				if (inst->internal.receive_timer >= RECEIVE_TIMEOUT)
				{
					NewLogEntry("ERR: Request timed out", inst->log);
					inst->status = ERROR_TIMEOUT_REQ;
					inst->last_error = ERROR_TIMEOUT_REQ;
					inst->internal.step = CREATE_REQUEST;
					break;
				}
			}
			else inst->internal.step = CLOSE_PORT;
			if(inst->internal.tcp_receive.status != tcpERR_NO_DATA)	inst->status = inst->internal.tcp_receive.status;
			else													inst->status = 0;
		break;
		/* ------------------------------------------------------------------------------------------ */
		/* Close connection */
		case CLOSE_PORT:
			inst->internal.tcp_close.enable 	= 1;
			inst->internal.tcp_close.ident		= inst->internal.tcp_open.ident;
			inst->internal.tcp_close.how 		= 0;
			TcpClose(&inst->internal.tcp_close);
			/* -------------------------------------------------------------------------------------- */
			/* Success */
			if(inst->internal.tcp_close.status == 0)
			{
				NewLogEntry("Port closed", inst->log);
				inst->internal.send_timer[0] = 0;
				inst->internal.step = WAIT;
			}
			else if(inst->internal.tcp_close.status == tcpERR_INVALID_IDENT)
			{
				inst->internal.step = ERROR;
			}
			inst->status = inst->internal.tcp_close.status;
		break;
		/* ------------------------------------------------------------------------------------------ */
		/* Wait before reopen port */
		case WAIT:
			inst->internal.tcp_open.enable = 0;
			TcpOpen(&inst->internal.tcp_open);
			inst->internal.tcp_client.enable = 0;
			TcpClient(&inst->internal.tcp_client);

			inst->internal.send_timer[0] += inst->cycle_time;
			if (inst->internal.send_timer[0] > 1000) inst->internal.step = OPEN_PORT;
		break;
		/* ------------------------------------------------------------------------------------------ */
		/* Error state */
		case ERROR:
			if (inst->status < 50000) inst->status = ERROR_CRITICAL;
			if (inst->enable == 0) inst->internal.step = DISABLE;
		break;
	}
}

/* ------------------------------------------------------------------------------------------------- */
/* Create new request to slave */
/* ------------------------------------------------------------------------------------------------- */
UINT create_request_to_slave(modbus_master_cfg_typ* config, USINT 	req_nr,	USINT* send_buff, UINT size_buf, UINT transaction_id, modbus_log_typ LOGBOOK)
{
	UINT	uint_var;
	INT		int_var;
	INT		value;
	UINT	data_len, i;

	/* Error message for undefined function code */
	memset(send_buff, 0, size_buf);
	/* Transaction id: 2 byte */
	uint_var = MySwapUINT(transaction_id);
	memcpy(&send_buff[0], &uint_var, sizeof(uint_var));
	/* Protocol id: 2 byte */
	uint_var = 0;
	memcpy(&send_buff[2], &uint_var, sizeof(uint_var));
	/* Length: 2 byte */
	/* Unit: 1 byte */
	send_buff[6] = (*config).action_param[req_nr].unit;
	switch((*config).action_param[req_nr].type)
	{
		case READ_COILS:
			/* Function code: 1 byte */
			send_buff[7] = READ_COILS;
			/* Strating address: 2 byte */
			uint_var = MySwapUINT((*config).action_param[req_nr].start_addr);
			memcpy(&send_buff[8], &uint_var, sizeof(uint_var));
			/* Coils number: 2 byte */
			uint_var = MySwapUINT((*config).action_param[req_nr].quantity);
			memcpy(&send_buff[10], &uint_var, sizeof(uint_var));
			/* Data len */
			data_len = 6;
			break;
		case READ_DISCRETE_INPUTS:
			/* Function code: 1 byte */
			send_buff[7] = READ_DISCRETE_INPUTS;
			/* Starting address: 2 byte */
			uint_var = MySwapUINT((*config).action_param[req_nr].start_addr);
			memcpy(&send_buff[8], &uint_var, sizeof(uint_var));
			/* Inputs number: 2 byte */
			uint_var = MySwapUINT((*config).action_param[req_nr].quantity);
			memcpy(&send_buff[10], &uint_var, sizeof(uint_var));
			/* Data length */
			data_len = 6;
			break;
		case READ_HOLDING_REGISTERS:
			/* Function code: 1 byte */
			send_buff[7] = READ_HOLDING_REGISTERS;
			/* Starting address: 2 byte */
			uint_var = MySwapUINT((*config).action_param[req_nr].start_addr);
			memcpy(&send_buff[8], &uint_var, sizeof(uint_var));
			/* Holding registers number: 2 byte */
			uint_var = MySwapUINT((*config).action_param[req_nr].quantity);
			memcpy(&send_buff[10], &uint_var, sizeof(uint_var));
			/* Data length */
			data_len = 6;
			break;
		case READ_INPUT_REGISTERS:
			/* Function code: 1 byte */
			send_buff[7] = READ_INPUT_REGISTERS;
			/* Starting address: 2 byte */
			uint_var = MySwapUINT((*config).action_param[req_nr].start_addr);
			memcpy(&send_buff[8], &uint_var, sizeof(uint_var));
			/* Input registers number: 2 byte */
			uint_var = MySwapUINT((*config).action_param[req_nr].quantity);
			memcpy(&send_buff[10], &uint_var, sizeof(uint_var));
			/* Data length */
			data_len = 6;
			break;
		case WRITE_SINGLE_COIL:
			/* Function code: 1 byte */
			send_buff[7] = WRITE_SINGLE_COIL;
			/* Starting address: 2 byte */
			uint_var = MySwapUINT((*config).action_param[req_nr].start_addr);
			memcpy(&send_buff[8], &uint_var, sizeof(uint_var));
			/* Value: 2 byte */
			if(*((BOOL*)((*config).action_param[req_nr].p_pv)))	value = ON;
			else												value = OFF;
			int_var = MySwapINT(value);
			memcpy(&send_buff[10], &int_var, sizeof(int_var));
			/* Data length */
			data_len = 6;
			break;
		case WRITE_SINGLE_REGISTER:
			/* Function code: 1 byte */
			send_buff[7] = WRITE_SINGLE_REGISTER;
			/* Starting address: 2 byte */
			uint_var = MySwapUINT((*config).action_param[req_nr].start_addr);
			memcpy(&send_buff[8], &uint_var, sizeof(uint_var));
			/* Value: 2 byte */
			value = *((INT*)((*config).action_param[req_nr].p_pv));
			int_var = MySwapINT(value);
			memcpy(&send_buff[10], &int_var, sizeof(int_var));
			/* Data length */
			data_len = 6;
			break;
		case WRITE_MULTIPLE_COILS:
			/* Function code: 1 byte */
			send_buff[7] = WRITE_MULTIPLE_COILS;
			/* Starting address: 2 byte */
			uint_var = MySwapUINT((*config).action_param[req_nr].start_addr);
			memcpy(&send_buff[8], &uint_var, sizeof(uint_var));
			/* Quantity: 2 byte */
			uint_var = MySwapUINT((*config).action_param[req_nr].quantity);
			memcpy(&send_buff[10], &uint_var, sizeof(uint_var));
			/* Byte count: 1 byte */
			if( (*config).action_param[req_nr].quantity % 8)	send_buff[12] = ((*config).action_param[req_nr].quantity / 8) + 1;
			else												send_buff[12] = (*config).action_param[req_nr].quantity / 8;
			/* Coil value: x byte */
			for(i = 0; i < (*config).action_param[req_nr].quantity; i++)
			{
				if(	((BOOL*)((*config).action_param[req_nr].p_pv))[i])
					send_buff[13 + (i/8)] = send_buff[13 + (i/8)] | (USINT)(0x01 << (i%8));
				else
					send_buff[13 + (i/8)] = send_buff[13 + (i/8)] & (USINT)~(0x01 << (i%8));
			}
			/* Data length */
			data_len = 7 + send_buff[12];
			break;

		case WRITE_MULTIPLE_REGISTERS:
			/* Function code: 1 byte */
			send_buff[7] = WRITE_MULTIPLE_REGISTERS;
			/* Starting address: 2 byte */
			uint_var = MySwapUINT((*config).action_param[req_nr].start_addr);
			memcpy(&send_buff[8], &uint_var, sizeof(uint_var));
			/* Quantity: 2 byte */
			uint_var = MySwapUINT((*config).action_param[req_nr].quantity);
			memcpy(&send_buff[10], &uint_var, sizeof(uint_var));
			/* Byte count: 1 byte */
			send_buff[12] = (*config).action_param[req_nr].quantity * 2;
			/* Coil value: x byte */
			for(i = 0; i < (*config).action_param[req_nr].quantity; i++)
			{
				value = ((INT*)((*config).action_param[req_nr].p_pv))[i];
				int_var = MySwapINT(value);
				memcpy(&send_buff[13 + (i*2)], &int_var, sizeof(int_var));
			}
			/* Data length */
			data_len = 7 + send_buff[12];
			break;

		default:
			/* Unsupported function code */
			NewLogEntry("ERR: Client function code", LOGBOOK);
			break;
	}
	/* Create log entry */
	MessageLog (TYP_REQUEST, (*config).action_param[req_nr].type, (*config).action_param[req_nr].start_addr, (*config).action_param[req_nr].quantity, LOGBOOK);

	/* Length: 2 byte */
	uint_var = MySwapUINT(data_len);
	memcpy(&send_buff[4], &uint_var, sizeof(uint_var));
	return 6 + data_len;
}

/* ------------------------------------------------------------------------------------------------- */
/* Analyse response from slave */
/* ------------------------------------------------------------------------------------------------- */
UINT analyze_answer_from_slave(modbus_master_cfg_typ* config,USINT req_nr, USINT* receive_buff, UINT transaction_id, modbus_log_typ LOGBOOK)
{
	INT		int_var;
	UINT	uint_var, receive_tr_id, protocol_id, length;
	UINT	unit, function_code, quantity, i;

	memcpy(&uint_var, &(receive_buff[0]), sizeof(uint_var));
	receive_tr_id	= MySwapUINT(uint_var);
	memcpy(&uint_var, &(receive_buff[2]), sizeof(uint_var));
	protocol_id		= MySwapUINT(uint_var);
	memcpy(&uint_var, &(receive_buff[4]), sizeof(uint_var));
	length 			= MySwapUINT(uint_var);
	unit 			= receive_buff[6];
	function_code	= receive_buff[7];

	if((receive_tr_id 	== transaction_id)	&&
	   (protocol_id		== 0)				&&
	   (length			> 0)				&&
	   (function_code	< 0x80))
	{
		switch(function_code)
		{
			case READ_COILS:
				/* Quantity: 1 byte */
				quantity = (*config).action_param[req_nr].quantity;
				/* Coil value: x byte */
				for(i = 0; i < quantity; i++)
				{
					if (receive_buff[9 + (i/8)] & (USINT)(0x01 << (i%8))) 	((BOOL*)((*config).action_param[req_nr].p_pv))[i] = 1;
					else													((BOOL*)((*config).action_param[req_nr].p_pv))[i] = 0;
				}
				break;

			case READ_DISCRETE_INPUTS:
				/* Quantity: 1 byte */
				quantity = (*config).action_param[req_nr].quantity;
				/* Coil value: x byte */
				for(i = 0; i < quantity; i++)
				{
					if (receive_buff[9 + (i/8)] & (USINT)(0x01 << (i%8)))	((BOOL*)((*config).action_param[req_nr].p_pv))[i] = 1;
					else													((BOOL*)((*config).action_param[req_nr].p_pv))[i] = 0;
				}
				break;

			case READ_HOLDING_REGISTERS:
				/* Quantity: 1 byte */
				quantity = receive_buff[8] / 2;
				/* Coil value: x byte */
				for(i = 0; i < quantity; i++)
				{
					memcpy(&int_var, &receive_buff[9 + (i*2)], sizeof(int_var));
					((INT*)((*config).action_param[req_nr].p_pv))[i] = MySwapINT(int_var);
				}
				break;

			case READ_INPUT_REGISTERS:
				/* Quantity: 1 byte */
				quantity = receive_buff[8] / 2;
				/* Coil value: x byte */
				for(i = 0; i < quantity; i++)
				{
					memcpy(&int_var, &receive_buff[9 + (i*2)], sizeof(int_var));
					((INT*)((*config).action_param[req_nr].p_pv))[i] = MySwapINT(int_var);
				}
				break;

			default:
				/* Unsupported function code */
				if ((function_code > WRITE_SINGLE_REGISTER) && ((function_code != WRITE_MULTIPLE_COILS) && (function_code != WRITE_MULTIPLE_REGISTERS)))
					NewLogEntry("ERR: Server function code", LOGBOOK);
				break;
		}
		/* Create log entry */
		MessageLog (TYP_RESPONSE, function_code, 0, 0, LOGBOOK);
	}
	/* Generate error on function exception from slave */
	else if(function_code >= 0x80)
	{
		function_code -= 0x80;
		switch(receive_buff[8])
			{
				case 1: NewLogEntry("ERR: Server->Bad function", LOGBOOK); break;
				case 2: NewLogEntry("ERR: Server->Data address", LOGBOOK); break;
				case 3: NewLogEntry("ERR: Server->Data value", LOGBOOK); break;
				case 4: NewLogEntry("ERR: Server->Device failure", LOGBOOK); break;
				case 5: NewLogEntry("ERR: Server->Exception ack", LOGBOOK); break;
				case 6: NewLogEntry("ERR: Server->Slave busy", LOGBOOK); break;
				case 10: NewLogEntry("ERR: Server->Path unavailable", LOGBOOK); break;
				default: NewLogEntry("ERR: Server->unknown", LOGBOOK); break;
			}
		return 1;
	}
	else
	{
		NewLogEntry("ERR: Bad slave message", LOGBOOK);
		return 1;
	}
	return 0;
}
```
